C05478=1134.009,150.819,-59.424,-178.763,7.145,148.974
C05479=1134.004,151.068,-59.444,-178.760,7.148,148.974
C05480=1133.999,151.317,-59.466,-178.758,7.150,148.974
C05481=1133.994,151.566,-59.487,-178.755,7.152,148.973
C05482=1133.989,151.815,-59.509,-178.752,7.154,148.973
C05483=1133.985,152.064,-59.529,-178.749,7.156,148.973
C05484=1133.980,152.313,-59.551,-178.746,7.158,148.972
C05485=1133.975,152.562,-59.572,-178.744,7.160,148.972
C05486=1133.970,152.811,-59.594,-178.741,7.162,148.972
C05487=1133.966,153.061,-59.615,-178.738,7.165,148.971
C05488=1133.962,153.309,-59.636,-178.735,7.166,148.971
C05489=1133.957,153.558,-59.657,-178.732,7.168,148.971
C05490=1133.952,153.807,-59.679,-178.729,7.171,148.970
C05491=1133.947,154.057,-59.700,-178.727,7.173,148.970
C05492=1133.942,154.306,-59.722,-178.723,7.175,148.970
C05493=1133.938,154.554,-59.743,-178.721,7.177,148.969
C05494=1133.934,154.804,-59.764,-178.718,7.179,148.969
C05495=1133.929,155.053,-59.786,-178.715,7.181,148.969
C05496=1133.923,155.302,-59.807,-178.712,7.183,148.968
C05497=1133.919,155.550,-59.828,-178.709,7.186,148.968
C05498=1133.914,155.800,-59.851,-178.707,7.188,148.968
C05499=1133.909,156.049,-59.871,-178.704,7.189,148.967
C05500=1133.904,156.298,-59.893,-178.701,7.192,148.967
C05501=1133.900,156.547,-59.915,-178.698,7.194,148.967
C05502=1133.896,156.795,-59.936,-178.695,7.196,148.967
C05503=1133.890,157.065,-59.960,-178.692,7.198,148.966
C05504=1133.885,157.334,-59.983,-178.689,7.201,148.966
C05505=1133.881,157.603,-60.006,-178.686,7.203,148.965
C05506=1133.875,157.872,-60.030,-178.683,7.205,148.965
C05507=1133.870,158.121,-60.052,-178.680,7.207,148.965
C05508=1133.866,158.371,-60.073,-178.678,7.209,148.965
C05509=1133.861,158.619,-60.095,-178.675,7.211,148.964
C05510=1133.856,158.868,-60.116,-178.672,7.214,148.964
C05511=1133.852,159.117,-60.138,-178.669,7.215,148.963
C05512=1133.847,159.366,-60.160,-178.666,7.218,148.963
C05513=1133.842,159.615,-60.182,-178.663,7.220,148.963
C05514=1133.838,159.864,-60.204,-178.660,7.223,148.963
C05515=1133.832,160.113,-60.225,-178.658,7.225,148.962
C05516=1133.828,160.362,-60.247,-178.655,7.226,148.962
C05517=1133.823,160.611,-60.268,-178.652,7.229,148.962
C05518=1133.819,160.860,-60.290,-178.649,7.231,148.961
C05519=1133.814,161.109,-60.312,-178.646,7.233,148.961
C05520=1133.810,161.358,-60.334,-178.643,7.235,148.961
C05521=1133.805,161.607,-60.356,-178.640,7.238,148.960
C05522=1133.800,161.856,-60.378,-178.638,7.240,148.960
C05523=1133.796,162.105,-60.400,-178.635,7.241,148.960
C05524=1133.791,162.354,-60.421,-178.632,7.244,148.959
C05525=1133.787,162.603,-60.443,-178.629,7.246,148.959
C05526=1133.782,162.852,-60.465,-178.626,7.248,148.959
C05527=1133.778,163.101,-60.487,-178.624,7.250,148.959
C05528=1133.772,163.350,-60.509,-178.620,7.253,148.958
C05529=1133.768,163.599,-60.531,-178.618,7.255,148.958
C05530=1133.763,163.848,-60.553,-178.615,7.257,148.958
C05531=1133.759,164.097,-60.575,-178.612,7.259,148.957
C05532=1133.754,164.346,-60.597,-178.609,7.262,148.957
C05533=1133.749,164.595,-60.619,-178.607,7.264,148.957
C05534=1133.745,164.844,-60.641,-178.604,7.265,148.956
C05535=1133.740,165.093,-60.664,-178.601,7.268,148.956
C05536=1133.735,165.341,-60.686,-178.598,7.270,148.956
C05537=1133.731,165.591,-60.708,-178.595,7.272,148.956
C05538=1133.726,165.839,-60.729,-178.593,7.274,148.955
C05539=1133.721,166.089,-60.752,-178.589,7.277,148.955
C05540=1133.716,166.338,-60.774,-178.587,7.279,148.955
C05541=1133.712,166.586,-60.796,-178.584,7.282,148.955
C05542=1133.707,166.835,-60.818,-178.581,7.283,148.954
C05543=1133.702,167.085,-60.841,-178.578,7.286,148.954
C05544=1133.698,167.334,-60.863,-178.576,7.288,148.954
C05545=1133.693,167.583,-60.884,-178.572,7.290,148.953
C05546=1133.689,167.831,-60.907,-178.570,7.292,148.953
C05547=1133.683,168.080,-60.929,-178.567,7.295,148.953
C05548=1133.679,168.330,-60.952,-178.564,7.297,148.952
C05549=1133.675,168.578,-60.974,-178.561,7.299,148.952
C05550=1133.670,168.827,-60.997,-178.559,7.301,148.952
C05551=1133.665,169.077,-61.019,-178.555,7.304,148.952
C05552=1133.661,169.325,-61.041,-178.553,7.306,148.951
C05553=1133.656,169.574,-61.064,-178.550,7.308,148.951
C05554=1133.651,169.823,-61.085,-178.547,7.310,148.951
C05555=1133.647,170.072,-61.108,-178.544,7.313,148.950
C05556=1133.642,170.321,-61.131,-178.542,7.315,148.950
C05557=1133.637,170.570,-61.152,-178.538,7.317,148.950
C05558=1133.633,170.819,-61.175,-178.536,7.319,148.950
C05559=1133.627,171.068,-61.197,-178.533,7.322,148.949
C05560=1133.624,171.316,-61.220,-178.530,7.324,148.949
C05561=1133.619,171.566,-61.243,-178.527,7.326,148.949
C05562=1133.614,171.814,-61.265,-178.524,7.328,148.948
C05563=1133.610,172.064,-61.287,-178.521,7.331,148.948
C05564=1133.605,172.313,-61.310,-178.519,7.333,148.948
C05565=1133.600,172.561,-61.332,-178.516,7.335,148.948
C05566=1133.595,172.811,-61.355,-178.513,7.337,148.947
C05567=1133.591,173.060,-61.378,-178.510,7.340,148.947
C05568=1133.586,173.308,-61.401,-178.507,7.342,148.947
C05569=1133.582,173.557,-61.423,-178.505,7.344,148.947
C05570=1133.577,173.806,-61.446,-178.501,7.347,148.946
C05571=1133.572,174.055,-61.468,-178.499,7.349,148.946
C05572=1133.567,174.304,-61.491,-178.496,7.352,148.946
C05573=1133.563,174.553,-61.513,-178.493,7.353,148.945
C05574=1133.558,174.802,-61.537,-178.490,7.356,148.945
C05575=1133.554,175.050,-61.559,-178.487,7.358,148.945
C05576=1133.549,175.300,-61.582,-178.485,7.361,148.945
C05577=1133.545,175.549,-61.604,-178.482,7.362,148.944
C05578=1133.540,175.798,-61.628,-178.479,7.365,148.944
C05579=1133.535,176.046,-61.649,-178.476,7.368,148.944
C05580=1133.531,176.295,-61.673,-178.473,7.370,148.944
C05581=1133.527,176.544,-61.696,-178.470,7.372,148.943
C05582=1133.522,176.794,-61.718,-178.468,7.374,148.943
C05583=1133.516,177.042,-61.741,-178.464,7.377,148.943
C05584=1133.512,177.291,-61.764,-178.462,7.379,148.943
C05585=1133.507,177.540,-61.787,-178.459,7.381,148.942
C05586=1133.503,177.789,-61.809,-178.456,7.384,148.942
C05587=1133.498,178.038,-61.832,-178.453,7.386,148.942
C05588=1133.493,178.287,-61.856,-178.450,7.389,148.942
C05589=1133.489,178.535,-61.879,-178.448,7.391,148.941
C05590=1133.484,178.785,-61.901,-178.445,7.393,148.941
C05591=1133.481,179.020,-61.923,-178.442,7.395,148.941
C05592=1133.476,179.256,-61.945,-178.439,7.398,148.941
C05593=1133.471,179.491,-61.967,-178.437,7.400,148.940
C05594=1133.449,180.668,-62.075,-179.293,9.081,149.576
C05595=1133.445,180.917,-62.098,-179.289,9.084,149.576
C05596=1133.440,181.165,-62.123,-179.286,9.087,149.576
C05597=1133.435,181.415,-62.146,-179.283,9.091,149.575
C05598=1133.431,181.664,-62.169,-179.280,9.094,149.575
C05599=1133.427,181.912,-62.192,-179.277,9.098,149.576
C05600=1133.422,182.161,-62.216,-179.274,9.100,149.575
C05601=1133.418,182.410,-62.239,-179.271,9.104,149.575
C05602=1133.413,182.659,-62.263,-179.268,9.107,149.575
C05603=1133.409,182.907,-62.287,-179.266,9.110,149.575
C05604=1133.404,183.156,-62.310,-179.262,9.114,149.575
C05605=1133.399,183.405,-62.334,-179.259,9.117,149.575
C05606=1133.395,183.654,-62.358,-179.257,9.120,149.575
C05607=1133.391,183.903,-62.381,-179.254,9.123,149.575
C05608=1133.386,184.152,-62.405,-179.251,9.127,149.575
C05609=1133.382,184.401,-62.429,-179.248,9.130,149.575
C05610=1133.377,184.650,-62.452,-179.246,9.133,149.575
C05611=1133.370,184.985,-62.485,-179.243,9.137,149.575
C05612=1133.364,185.319,-62.516,-179.238,9.141,149.575
C05613=1133.358,185.653,-62.548,-179.235,9.145,149.575
C05614=1133.352,185.987,-62.581,-179.232,9.149,149.575
C05615=1133.347,186.236,-62.604,-179.230,9.152,149.575
C05616=1133.343,186.485,-62.628,-179.227,9.154,149.575
C05617=1133.339,186.734,-62.652,-179.224,9.158,149.575
C05618=1133.334,186.983,-62.676,-179.222,9.161,149.575
C05619=1133.329,187.232,-62.700,-179.220,9.163,149.575
C05620=1133.325,187.481,-62.724,-179.217,9.166,149.575
C05621=1133.320,187.730,-62.747,-179.215,9.169,149.575
C05622=1133.315,187.978,-62.771,-179.212,9.172,149.575
C05623=1133.311,188.226,-62.795,-179.210,9.175,149.575
C05624=1133.306,188.475,-62.819,-179.208,9.178,149.575
C05625=1133.302,188.725,-62.844,-179.206,9.180,149.575
C05626=1133.297,188.974,-62.867,-179.203,9.183,149.575
C05627=1133.293,189.222,-62.891,-179.201,9.186,149.576
C05628=1133.288,189.471,-62.915,-179.199,9.189,149.576
C05629=1133.284,189.720,-62.939,-179.197,9.191,149.576
C05630=1133.279,189.968,-62.963,-179.194,9.194,149.576
C05631=1133.275,190.218,-62.988,-179.192,9.196,149.576
C05632=1133.270,190.466,-63.012,-179.191,9.199,149.576
C05633=1133.266,190.715,-63.035,-179.188,9.202,149.576
C05634=1133.261,190.964,-63.060,-179.187,9.205,149.576
C05635=1133.256,191.212,-63.084,-179.185,9.207,149.576
C05636=1133.251,191.461,-63.107,-179.183,9.210,149.576
C05637=1133.248,191.710,-63.132,-179.181,9.213,149.576
C05638=1133.243,191.959,-63.156,-179.179,9.215,149.576
C05639=1133.238,192.207,-63.180,-179.177,9.218,149.577
C05640=1133.234,192.456,-63.204,-179.175,9.220,149.577
C05641=1133.229,192.706,-63.229,-179.174,9.222,149.577
C05642=1133.224,192.954,-63.253,-179.172,9.225,149.577
C05643=1133.220,193.203,-63.277,-179.170,9.227,149.577
C05644=1133.215,193.451,-63.302,-179.169,9.230,149.577
C05645=1133.211,193.700,-63.326,-179.167,9.232,149.577
C05646=1133.206,193.950,-63.349,-179.165,9.235,149.577
C05647=1133.201,194.198,-63.374,-179.164,9.238,149.578
C05648=1133.197,194.447,-63.398,-179.162,9.240,149.578
C05649=1133.193,194.695,-63.422,-179.161,9.243,149.578
C05650=1133.188,194.945,-63.447,-179.159,9.246,149.578
C05651=1133.184,195.193,-63.471,-179.158,9.247,149.578
C05652=1133.179,195.441,-63.495,-179.156,9.250,149.578
C05653=1133.174,195.690,-63.520,-179.155,9.253,149.579
C05654=1133.170,195.939,-63.544,-179.153,9.255,149.579
C05655=1133.166,196.188,-63.568,-179.153,9.257,149.579
C05656=1133.160,196.437,-63.593,-179.148,9.261,149.579
C05657=1133.157,196.686,-63.617,-179.144,9.266,149.579
C05658=1133.152,196.935,-63.642,-179.140,9.269,149.579
C05659=1133.147,197.183,-63.666,-179.136,9.273,149.578
C05660=1133.143,197.432,-63.690,-179.132,9.277,149.578
C05661=1133.138,197.681,-63.715,-179.128,9.281,149.578
C05662=1133.134,197.929,-63.739,-179.123,9.285,149.578
C05663=1133.129,198.144,-63.761,-179.120,9.288,149.578
C05664=1133.126,198.358,-63.782,-179.117,9.291,149.577
C05665=1133.122,198.572,-63.803,-179.113,9.295,149.577
C05666=1133.118,198.787,-63.824,-179.110,9.298,149.577
C05667=1133.115,199.002,-63.845,-179.107,9.301,149.577
C05668=1133.110,199.216,-63.867,-179.103,9.304,149.577
C05669=1133.106,199.431,-63.888,-179.100,9.307,149.577
C05670=1133.103,199.645,-63.909,-179.097,9.311,149.577
C05671=1133.098,199.894,-63.934,-179.093,9.314,149.576
C05672=1133.094,200.143,-63.959,-179.089,9.318,149.576
C05673=1133.089,200.392,-63.983,-179.085,9.321,149.576
C05674=1133.085,200.639,-64.008,-179.082,9.324,149.576
C05675=1133.080,200.889,-64.033,-179.078,9.328,149.576
C05676=1133.075,201.138,-64.058,-179.075,9.331,149.576
C05677=1133.071,201.387,-64.082,-179.071,9.335,149.575
C05678=1133.066,201.635,-64.108,-179.068,9.338,149.575
C05679=1133.063,201.884,-64.132,-179.065,9.341,149.575
C05680=1133.058,202.133,-64.157,-179.061,9.345,149.575
C05681=1133.053,202.381,-64.182,-179.058,9.347,149.575
C05682=1133.049,202.630,-64.206,-179.054,9.351,149.575
C05683=1133.045,202.879,-64.232,-179.051,9.354,149.575
C05684=1133.040,203.127,-64.257,-179.048,9.357,149.574
C05685=1133.035,203.376,-64.281,-179.045,9.360,149.574
C05686=1133.031,203.625,-64.307,-179.041,9.363,149.574
C05687=1133.026,203.873,-64.331,-179.038,9.366,149.574
C05688=1133.022,204.122,-64.357,-179.035,9.369,149.574
C05689=1133.017,204.370,-64.381,-179.033,9.372,149.574
C05690=1133.013,204.619,-64.407,-179.029,9.375,149.574
C05691=1133.008,204.868,-64.432,-179.026,9.378,149.574
C05692=1133.004,205.117,-64.457,-179.023,9.381,149.573
C05693=1133.000,205.366,-64.482,-179.020,9.384,149.573
C05694=1132.995,205.614,-64.507,-179.018,9.387,149.573
C05695=1132.990,205.863,-64.532,-179.015,9.390,149.573
C05696=1132.986,206.112,-64.558,-179.012,9.392,149.573
C05697=1132.981,206.360,-64.583,-179.010,9.395,149.573
C05698=1132.976,206.609,-64.608,-179.007,9.397,149.573
C05699=1132.973,206.858,-64.633,-179.005,9.401,149.573
C05700=1132.968,207.106,-64.658,-179.002,9.403,149.573
C05701=1132.963,207.355,-64.684,-179.000,9.406,149.573
C05702=1132.959,207.604,-64.709,-178.997,9.408,149.573
C05703=1132.954,207.853,-64.734,-178.995,9.411,149.573
C05704=1132.950,208.101,-64.760,-178.992,9.414,149.573
C05705=1132.945,208.350,-64.785,-178.991,9.416,149.573
C05706=1132.940,208.599,-64.810,-178.988,9.419,149.573
C05707=1132.936,208.847,-64.835,-178.986,9.421,149.573
C05708=1132.932,209.096,-64.861,-178.984,9.423,149.573
C05709=1132.928,209.344,-64.886,-178.981,9.427,149.573
C05710=1132.923,209.593,-64.911,-178.979,9.429,149.573
C05711=1132.919,209.842,-64.937,-178.978,9.431,149.573
C05712=1132.914,210.091,-64.963,-178.976,9.434,149.573
C05713=1132.910,210.339,-64.988,-178.974,9.436,149.573
C05714=1132.905,210.588,-65.013,-178.972,9.439,149.573
C05715=1132.900,210.836,-65.038,-178.970,9.441,149.573
C05716=1132.896,211.085,-65.064,-178.968,9.443,149.573
C05717=1132.892,211.334,-65.090,-178.967,9.446,149.574
C05718=1132.887,211.582,-65.115,-178.965,9.448,149.574
C05719=1132.884,211.797,-65.137,-178.963,9.451,149.574
C05720=1132.880,212.011,-65.159,-178.962,9.453,149.574
C05721=1132.875,212.225,-65.181,-178.960,9.455,149.574
C05722=1132.872,212.440,-65.203,-178.960,9.457,149.574
C05723=1132.868,212.654,-65.225,-178.958,9.458,149.574
C05724=1132.864,212.868,-65.247,-178.957,9.461,149.575
C05725=1132.860,213.083,-65.269,-178.956,9.463,149.575
C05726=1132.856,213.297,-65.291,-178.955,9.465,149.575
C05727=1132.852,213.546,-65.317,-178.953,9.467,149.575
C05728=1132.847,213.794,-65.342,-178.952,9.470,149.575
C05729=1132.843,214.043,-65.368,-178.950,9.472,149.575
C05730=1132.839,214.292,-65.394,-178.948,9.476,149.576
C05731=1132.834,214.540,-65.419,-178.946,9.478,149.576
C05732=1132.830,214.789,-65.445,-178.944,9.481,149.576
C05733=1132.825,215.038,-65.471,-178.943,9.483,149.576
C05734=1132.821,215.286,-65.496,-178.940,9.487,149.576
C05735=1132.816,215.535,-65.522,-178.939,9.489,149.576
C05736=1132.812,215.783,-65.548,-178.937,9.492,149.576
C05737=1132.808,216.032,-65.573,-178.935,9.495,149.577
C05738=1132.803,216.280,-65.599,-178.933,9.497,149.577
C05739=1132.799,216.529,-65.625,-178.931,9.501,149.577
C05740=1132.795,216.778,-65.650,-178.929,9.503,149.577
C05741=1132.790,217.026,-65.676,-178.927,9.506,149.577
C05742=1132.785,217.275,-65.702,-178.925,9.509,149.577
C05743=1132.781,217.524,-65.728,-178.922,9.512,149.577
C05744=1132.776,217.773,-65.754,-178.920,9.515,149.577
C05745=1132.772,218.021,-65.779,-178.918,9.518,149.578
C05746=1132.767,218.270,-65.805,-178.916,9.521,149.578
C05747=1132.763,218.518,-65.830,-178.914,9.524,149.578
C05748=1132.759,218.767,-65.856,-178.911,9.527,149.578
C05749=1132.754,219.016,-65.883,-178.908,9.530,149.578
C05750=1132.749,219.264,-65.909,-178.906,9.533,149.578
C05751=1132.745,219.513,-65.934,-178.903,9.537,149.578
C05752=1132.741,219.761,-65.960,-178.901,9.540,149.578
C05753=1132.737,220.010,-65.986,-178.898,9.543,149.578
C05754=1132.732,220.259,-66.012,-178.896,9.546,149.578
C05755=1132.727,220.507,-66.038,-178.893,9.549,149.578
C05756=1132.723,220.756,-66.064,-178.891,9.552,149.578
C05757=1132.719,221.004,-66.090,-178.888,9.555,149.578
C05758=1132.714,221.254,-66.116,-178.886,9.558,149.579
C05759=1132.710,221.502,-66.142,-178.883,9.561,149.579
C05760=1132.705,221.750,-66.168,-178.880,9.565,149.579
C05761=1132.701,221.999,-66.194,-178.877,9.568,149.579
C05762=1132.696,222.248,-66.220,-178.875,9.572,149.579
C05763=1132.692,222.496,-66.247,-178.872,9.575,149.579
C05764=1132.688,222.745,-66.272,-178.869,9.578,149.579
C05765=1132.683,222.994,-66.299,-178.866,9.581,149.579
C05766=1132.679,223.242,-66.325,-178.863,9.585,149.579
C05767=1132.674,223.490,-66.351,-178.860,9.588,149.579
C05768=1132.669,223.739,-66.378,-178.857,9.592,149.579
C05769=1132.665,223.987,-66.403,-178.855,9.595,149.579
C05770=1132.661,224.236,-66.429,-178.851,9.598,149.579
C05771=1132.656,224.485,-66.456,-178.848,9.601,149.579
C05772=1132.652,224.734,-66.482,-178.845,9.605,149.579
C05773=1132.648,224.982,-66.508,-178.842,9.609,149.579
C05774=1132.643,225.231,-66.535,-178.838,9.612,149.579
C05775=1132.639,225.445,-66.558,-178.836,9.616,149.579
C05776=1132.636,225.659,-66.581,-178.833,9.618,149.579
C05777=1132.631,225.873,-66.603,-178.830,9.621,149.578
C05778=1132.628,226.088,-66.626,-178.827,9.624,149.578
C05779=1132.624,226.301,-66.649,-178.824,9.627,149.578
C05780=1132.620,226.516,-66.671,-178.821,9.630,149.578
C05781=1132.616,226.730,-66.694,-178.818,9.633,149.578
C05782=1132.613,226.944,-66.717,-178.815,9.636,149.578
C05783=1132.608,227.193,-66.743,-178.812,9.640,149.578
C05784=1132.604,227.441,-66.770,-178.808,9.643,149.578
C05785=1132.600,227.690,-66.796,-178.804,9.647,149.578
C05786=1132.595,227.939,-66.823,-178.801,9.650,149.578
C05787=1132.591,228.187,-66.849,-178.797,9.654,149.578
C05788=1132.586,228.435,-66.876,-178.794,9.657,149.577
C05789=1132.582,228.684,-66.902,-178.790,9.661,149.577
C05790=1132.577,228.933,-66.929,-178.786,9.664,149.577
C05791=1132.573,229.181,-66.956,-178.782,9.668,149.577
C05792=1132.569,229.429,-66.983,-178.778,9.672,149.577
C05793=1132.564,229.679,-67.009,-178.775,9.675,149.577
C05794=1132.560,229.927,-67.035,-178.771,9.679,149.576
C05795=1132.555,230.175,-67.062,-178.766,9.683,149.576
C05796=1132.551,230.424,-67.089,-178.762,9.686,149.576
C05797=1132.547,230.672,-67.116,-178.759,9.690,149.576
C05798=1132.542,230.920,-67.143,-178.755,9.693,149.576
C05799=1132.537,231.169,-67.170,-178.751,9.696,149.575
C05800=1132.534,231.418,-67.197,-178.748,9.700,149.575
C05801=1132.529,231.667,-67.223,-178.745,9.702,149.575
C05802=1132.524,231.915,-67.250,-178.741,9.706,149.575
C05803=1132.521,232.164,-67.277,-178.737,9.709,149.575
C05804=1132.516,232.412,-67.304,-178.734,9.713,149.575
C05805=1132.511,232.661,-67.331,-178.731,9.715,149.575
C05806=1132.507,232.909,-67.358,-178.727,9.719,149.574
C05807=1132.503,233.157,-67.384,-178.724,9.721,149.574
C05808=1132.499,233.406,-67.412,-178.720,9.725,149.574
C05809=1132.494,233.654,-67.440,-178.717,9.728,149.574
C05810=1132.490,233.903,-67.467,-178.714,9.731,149.574
C05811=1132.486,234.151,-67.493,-178.711,9.734,149.574
C05812=1132.481,234.399,-67.520,-178.708,9.737,149.573
C05813=1132.476,234.648,-67.547,-178.704,9.740,149.573
C05814=1132.472,234.897,-67.575,-178.701,9.742,149.573
C05815=1132.468,235.146,-67.602,-178.698,9.745,149.573
C05816=1132.463,235.394,-67.629,-178.695,9.748,149.573
C05817=1132.459,235.642,-67.656,-178.692,9.751,149.573
C05818=1132.455,235.890,-67.683,-178.689,9.753,149.573
C05819=1132.451,236.139,-67.711,-178.686,9.756,149.572
C05820=1132.446,236.388,-67.738,-178.683,9.759,149.572
C05821=1132.441,236.636,-67.765,-178.681,9.762,149.572
C05822=1132.437,236.884,-67.792,-178.678,9.765,149.572
C05823=1132.433,237.133,-67.820,-178.675,9.768,149.572
C05824=1132.428,237.382,-67.847,-178.672,9.770,149.572
C05825=1132.424,237.630,-67.875,-178.669,9.772,149.572
C05826=1132.419,237.878,-67.902,-178.666,9.775,149.572
C05827=1132.416,238.127,-67.929,-178.665,9.777,149.572
C05828=1132.411,238.376,-67.956,-178.662,9.780,149.572
C05829=1132.407,238.624,-67.983,-178.659,9.782,149.571
C05830=1132.402,238.872,-68.010,-178.657,9.785,149.572
C05831=1132.398,239.086,-68.035,-178.654,9.787,149.571
C05832=1132.395,239.301,-68.058,-178.653,9.790,149.571
C05833=1132.391,239.515,-68.082,-178.650,9.791,149.571
C05834=1132.387,239.728,-68.105,-178.648,9.794,149.571
C05835=1132.383,239.943,-68.129,-178.647,9.795,149.571
C05836=1132.380,240.157,-68.153,-178.645,9.797,149.571
C05837=1132.376,240.371,-68.176,-178.643,9.800,149.571
C05838=1132.372,240.585,-68.201,-178.641,9.802,149.571
C05839=1132.368,240.834,-68.228,-178.639,9.804,149.571
C05840=1132.363,241.082,-68.255,-178.637,9.806,149.571
C05841=1132.359,241.331,-68.283,-178.634,9.808,149.571
C05842=1132.355,241.579,-68.310,-178.633,9.811,149.571
C05843=1132.350,241.827,-68.338,-178.631,9.813,149.571
C05844=1132.346,242.076,-68.365,-178.629,9.815,149.571
C05845=1132.342,242.324,-68.393,-178.627,9.818,149.571
C05846=1132.337,242.573,-68.420,-178.625,9.820,149.571
C05847=1132.334,242.821,-68.448,-178.623,9.822,149.572
C05848=1132.329,243.070,-68.475,-178.622,9.824,149.572
C05849=1132.325,243.317,-68.503,-178.620,9.826,149.572
C05850=1132.320,243.567,-68.531,-178.618,9.828,149.572
C05851=1132.315,243.815,-68.559,-178.617,9.830,149.572
C05852=1132.311,244.063,-68.587,-178.615,9.832,149.572
C05853=1132.307,244.312,-68.614,-178.613,9.835,149.572
C05854=1132.303,244.560,-68.642,-178.612,9.837,149.572
C05855=1132.298,244.808,-68.669,-178.610,9.839,149.572
C05856=1132.294,245.057,-68.697,-178.609,9.841,149.572
C05857=1132.290,245.305,-68.725,-178.607,9.843,149.572
C05858=1132.286,245.554,-68.752,-178.606,9.845,149.572
C05859=1132.281,245.802,-68.781,-178.605,9.847,149.573
C05860=1132.276,246.051,-68.808,-178.604,9.849,149.573
C05861=1132.272,246.299,-68.836,-178.603,9.851,149.573
C05862=1132.268,246.547,-68.863,-178.602,9.853,149.573
C05863=1132.263,246.796,-68.891,-178.601,9.855,149.573
C05864=1132.260,247.044,-68.919,-178.599,9.857,149.574
C05865=1132.254,247.292,-68.947,-178.598,9.859,149.574
C05866=1132.250,247.542,-68.974,-178.594,9.863,149.574
C05867=1132.246,247.789,-69.002,-178.586,9.869,149.573
C05868=1132.242,248.037,-69.030,-178.578,9.875,149.572
C05869=1132.238,248.286,-69.057,-178.571,9.880,149.572
C05870=1132.233,248.535,-69.086,-178.565,9.886,149.571
C05871=1132.229,248.783,-69.114,-178.557,9.891,149.571
C05872=1132.224,249.031,-69.142,-178.551,9.895,149.570
C05873=1132.221,249.280,-69.170,-178.545,9.900,149.569
C05874=1132.216,249.528,-69.198,-178.539,9.905,149.569
C05875=1132.212,249.776,-69.226,-178.533,9.909,149.569
C05876=1132.207,250.025,-69.255,-178.528,9.913,149.568
C05877=1132.203,250.273,-69.283,-178.523,9.917,149.568
C05878=1132.199,250.521,-69.311,-178.518,9.920,149.567
C05879=1132.194,250.770,-69.339,-178.513,9.924,149.567
C05880=1132.190,251.018,-69.367,-178.509,9.928,149.567
C05881=1132.185,251.267,-69.396,-178.505,9.931,149.566
C05882=1132.182,251.515,-69.424,-178.501,9.934,149.566
C05883=1132.177,251.763,-69.452,-178.498,9.936,149.566
C05884=1132.173,252.012,-69.481,-178.495,9.939,149.566
C05885=1132.168,252.260,-69.508,-178.491,9.942,149.565
C05886=1132.164,252.509,-69.537,-178.489,9.943,149.565
C05887=1132.160,252.723,-69.562,-178.487,9.945,149.565
C05888=1132.157,252.936,-69.586,-178.485,9.948,149.565
C05889=1132.153,253.150,-69.611,-178.483,9.949,149.565
C05890=1132.149,253.364,-69.635,-178.482,9.951,149.565
C05891=1132.146,253.578,-69.660,-178.481,9.952,149.565
C05892=1132.142,253.792,-69.684,-178.480,9.953,149.565
C05893=1132.138,254.006,-69.709,-178.479,9.954,149.565
C05894=1132.134,254.220,-69.733,-178.479,9.956,149.565
C05895=1132.131,254.468,-69.762,-178.478,9.956,149.565
C05896=1132.125,254.716,-69.790,-178.478,9.957,149.566
C05897=1132.122,254.965,-69.818,-178.479,9.958,149.566
C05898=1132.117,255.214,-69.847,-178.478,9.959,149.566
C05899=1132.113,255.462,-69.875,-178.479,9.960,149.567
C05900=1132.109,255.710,-69.904,-178.481,9.960,149.567
C05901=1132.104,255.958,-69.932,-178.481,9.961,149.567
C05902=1132.100,256.207,-69.961,-178.479,9.963,149.567
C05903=1132.096,256.455,-69.989,-178.476,9.966,149.567
C05904=1132.091,256.704,-70.017,-178.473,9.969,149.567
C05905=1132.088,256.952,-70.046,-178.470,9.972,149.567
C05906=1132.083,257.200,-70.075,-178.467,9.976,149.567
C05907=1132.078,257.449,-70.103,-178.464,9.978,149.567
C05908=1132.074,257.697,-70.131,-178.461,9.981,149.567
C05909=1132.069,257.945,-70.161,-178.458,9.984,149.567
C05910=1132.066,258.193,-70.189,-178.454,9.987,149.567
C05911=1132.061,258.442,-70.217,-178.451,9.990,149.566
C05912=1132.057,258.689,-70.246,-178.448,9.993,149.566
C05913=1132.053,258.938,-70.275,-178.444,9.996,149.566
C05914=1132.049,259.187,-70.304,-178.441,9.999,149.566
C05915=1132.045,259.435,-70.332,-178.438,10.002,149.566
C05916=1132.040,259.683,-70.361,-178.435,10.005,149.566
C05917=1132.036,259.932,-70.390,-178.431,10.008,149.565
C05918=1132.032,260.180,-70.418,-178.428,10.011,149.565
C05919=1132.027,260.428,-70.447,-178.424,10.015,149.565
C05920=1132.022,260.677,-70.476,-178.421,10.017,149.565
C05921=1132.019,260.925,-70.505,-178.417,10.021,149.565
C05922=1132.015,261.174,-70.534,-178.414,10.024,149.565
C05923=1132.010,261.421,-70.563,-178.410,10.026,149.564
C05924=1132.005,261.670,-70.591,-178.407,10.030,149.564
C05925=1132.002,261.918,-70.620,-178.403,10.033,149.564
C05926=1131.997,262.167,-70.649,-178.399,10.036,149.564
C05927=1131.993,262.414,-70.678,-178.396,10.039,149.564
C05928=1131.988,262.663,-70.708,-178.392,10.042,149.563
C05929=1131.985,262.911,-70.736,-178.388,10.045,149.563
C05930=1131.980,263.160,-70.765,-178.384,10.049,149.563
C05931=1131.975,263.408,-70.794,-178.380,10.052,149.563
C05932=1131.971,263.656,-70.823,-178.376,10.055,149.562
C05933=1131.967,263.904,-70.852,-178.372,10.058,149.562
C05934=1131.963,264.152,-70.882,-178.368,10.062,149.562
C05935=1131.959,264.401,-70.910,-178.364,10.065,149.562
C05936=1131.954,264.649,-70.939,-178.361,10.068,149.562
C05937=1131.950,264.897,-70.969,-178.359,10.070,149.561
C05938=1131.946,265.145,-70.998,-178.357,10.072,149.561
C05939=1131.941,265.394,-71.027,-178.354,10.074,149.561
C05940=1131.937,265.642,-71.056,-178.352,10.077,149.561
C05941=1131.933,265.891,-71.086,-178.350,10.079,149.561
C05942=1131.928,266.138,-71.115,-178.347,10.081,149.561
C05943=1131.925,266.353,-71.140,-178.344,10.083,149.561
C05944=1131.921,266.566,-71.165,-178.343,10.086,149.561
C05945=1131.918,266.780,-71.190,-178.341,10.087,149.561
C05946=1131.914,266.993,-71.216,-178.339,10.089,149.561
C05947=1131.910,267.208,-71.241,-178.336,10.091,149.561
C05948=1131.907,267.422,-71.266,-178.334,10.093,149.561
C05949=1131.903,267.635,-71.291,-178.332,10.095,149.560
C05950=1131.899,267.849,-71.317,-178.329,10.098,149.560
C05951=1131.894,268.098,-71.345,-178.327,10.100,149.560
C05952=1131.890,268.346,-71.375,-178.324,10.103,149.560
C05953=1131.886,268.594,-71.404,-178.322,10.105,149.560
C05954=1131.882,268.843,-71.434,-178.319,10.107,149.560
C05955=1131.878,269.091,-71.463,-178.317,10.110,149.560
C05956=1131.873,269.339,-71.493,-178.314,10.113,149.560
C05957=1131.869,269.587,-71.522,-178.311,10.115,149.560
C05958=1131.865,269.836,-71.552,-178.308,10.118,149.560
C05959=1131.861,270.084,-71.581,-178.306,10.120,149.560
C05960=1131.857,270.332,-71.611,-178.303,10.123,149.559
C05961=1131.853,270.580,-71.640,-178.300,10.126,149.559
C05962=1131.848,270.828,-71.669,-178.297,10.128,149.559
C05963=1131.844,271.076,-71.699,-178.295,10.130,149.559
C05964=1131.839,271.324,-71.728,-178.292,10.133,149.559
C05965=1131.836,271.572,-71.758,-178.289,10.136,149.559
C05966=1131.831,271.820,-71.788,-178.286,10.139,149.559
C05967=1131.827,272.069,-71.817,-178.282,10.141,149.559
C05968=1131.823,272.317,-71.847,-178.279,10.144,149.558
C05969=1131.819,272.565,-71.876,-178.276,10.146,149.558
C05970=1131.814,272.814,-71.906,-178.274,10.148,149.558
C05971=1131.810,273.062,-71.936,-178.271,10.151,149.558
C05972=1131.806,273.310,-71.966,-178.268,10.154,149.558
C05973=1131.802,273.558,-71.995,-178.265,10.157,149.558
C05974=1131.797,273.806,-72.025,-178.262,10.159,149.558
C05975=1131.793,274.055,-72.054,-178.259,10.162,149.558
C05976=1131.789,274.302,-72.085,-178.255,10.165,149.557
C05977=1131.785,274.551,-72.114,-178.253,10.168,149.557
C05978=1131.780,274.799,-72.144,-178.250,10.171,149.557
C05979=1131.776,275.047,-72.173,-178.246,10.173,149.557
C05980=1131.772,275.295,-72.203,-178.243,10.176,149.557
C05981=1131.768,275.544,-72.234,-178.240,10.179,149.557
C05982=1131.764,275.792,-72.263,-178.237,10.181,149.556
C05983=1131.760,276.040,-72.293,-178.234,10.184,149.556
C05984=1131.756,276.288,-72.323,-178.231,10.188,149.556
C05985=1131.751,276.537,-72.353,-178.227,10.190,149.556
C05986=1131.747,276.785,-72.383,-178.224,10.193,149.556
C05987=1131.743,277.033,-72.412,-178.221,10.195,149.556
C05988=1131.739,277.281,-72.443,-178.217,10.199,149.556
C05989=1131.734,277.529,-72.473,-178.214,10.201,149.555
C05990=1131.730,277.777,-72.502,-178.211,10.204,149.555
C05991=1131.726,278.025,-72.532,-178.207,10.207,149.555
C05992=1131.722,278.274,-72.563,-178.204,10.210,149.555
C05993=1131.718,278.522,-72.593,-178.201,10.212,149.554
C05994=1131.714,278.770,-72.622,-178.197,10.216,149.554
C05995=1131.709,279.018,-72.653,-178.194,10.218,149.554
C05996=1131.705,279.266,-72.683,-178.190,10.221,149.554
C05997=1131.701,279.514,-72.713,-178.187,10.224,149.554
C05998=1131.696,279.762,-72.744,-178.184,10.227,149.553
C05999=1131.693,279.976,-72.769,-178.181,10.229,149.553
C06000=1131.689,280.190,-72.795,-178.177,10.232,149.553
C06001=1131.686,280.404,-72.822,-178.174,10.234,149.553
C06002=1131.682,280.617,-72.847,-178.171,10.237,149.553
C06003=1131.679,280.831,-72.874,-178.168,10.240,149.553
C06004=1131.674,281.045,-72.900,-178.165,10.242,149.552
C06005=1131.672,281.258,-72.926,-178.162,10.244,149.552
C06006=1131.667,281.472,-72.952,-178.159,10.246,149.552
C06007=1131.663,281.720,-72.982,-178.156,10.249,149.552
C06008=1131.659,281.969,-73.012,-178.153,10.252,149.552
C06009=1131.655,282.217,-73.042,-178.150,10.254,149.551
C06010=1131.651,282.464,-73.073,-178.147,10.257,149.551
C06011=1131.647,282.712,-73.103,-178.144,10.260,149.551
C06012=1131.642,282.961,-73.133,-178.140,10.262,149.551
C06013=1131.639,283.209,-73.164,-178.137,10.265,149.551
C06014=1131.634,283.457,-73.195,-178.134,10.267,149.550
C06015=1131.629,283.705,-73.225,-178.131,10.270,149.550
C06016=1131.625,283.953,-73.256,-178.129,10.272,149.550
C06017=1131.621,284.202,-73.286,-178.125,10.274,149.550
C06018=1131.617,284.450,-73.316,-178.122,10.277,149.550
C06019=1131.613,284.697,-73.347,-178.119,10.279,149.550
C06020=1131.609,284.945,-73.377,-178.116,10.282,149.549
C06021=1131.605,285.194,-73.408,-178.113,10.285,149.549
C06022=1131.600,285.442,-73.439,-178.110,10.287,149.549
C06023=1131.596,285.689,-73.469,-178.107,10.290,149.549
C06024=1131.592,285.938,-73.500,-178.104,10.293,149.549
C06025=1131.588,286.186,-73.531,-178.101,10.295,149.549
C06026=1131.584,286.434,-73.561,-178.098,10.297,149.548
C06027=1131.579,286.682,-73.592,-178.095,10.300,149.548
C06028=1131.576,286.930,-73.622,-178.092,10.302,149.548
C06029=1131.571,287.178,-73.653,-178.089,10.305,149.548
C06030=1131.567,287.426,-73.684,-178.085,10.307,149.548
C06031=1131.563,287.674,-73.715,-178.082,10.310,149.547
C06032=1131.559,287.922,-73.745,-178.079,10.313,149.547
C06033=1131.554,288.170,-73.776,-178.076,10.315,149.547
C06034=1131.550,288.419,-73.807,-178.073,10.318,149.547
C06035=1131.546,288.666,-73.837,-178.070,10.320,149.547
C06036=1131.542,288.914,-73.868,-178.067,10.323,149.547
C06037=1131.538,289.163,-73.899,-178.064,10.326,149.546
C06038=1131.533,289.411,-73.930,-178.061,10.328,149.546
C06039=1131.530,289.659,-73.961,-178.058,10.330,149.546
C06040=1131.525,289.907,-73.992,-178.055,10.333,149.546
C06041=1131.521,290.155,-74.023,-178.052,10.335,149.546
C06042=1131.517,290.403,-74.054,-178.049,10.338,149.545
C06043=1131.513,290.651,-74.084,-178.045,10.340,149.545
C06044=1131.509,290.900,-74.115,-178.042,10.343,149.545
C06045=1131.505,291.147,-74.147,-178.040,10.346,149.545
C06046=1131.500,291.395,-74.177,-178.036,10.348,149.545
C06047=1131.496,291.644,-74.209,-178.033,10.351,149.545
C06048=1131.492,291.891,-74.239,-178.030,10.354,149.544
C06049=1131.488,292.139,-74.271,-178.027,10.356,149.544
C06050=1131.484,292.387,-74.301,-178.024,10.358,149.544
C06051=1131.480,292.636,-74.332,-178.021,10.361,149.544
C06052=1131.476,292.883,-74.364,-178.018,10.363,149.544
C06053=1131.471,293.131,-74.395,-178.015,10.366,149.544
C06054=1131.467,293.380,-74.426,-178.012,10.368,149.543
C06055=1131.463,293.594,-74.453,-178.009,10.370,149.543
C06056=1131.460,293.806,-74.480,-178.007,10.373,149.543
C06057=1131.456,294.020,-74.507,-178.004,10.375,149.543
C06058=1131.453,294.234,-74.534,-178.001,10.378,149.543
C06059=1131.449,294.447,-74.560,-177.999,10.380,149.543
C06060=1131.446,294.661,-74.587,-177.996,10.382,149.542
C06061=1131.442,294.875,-74.614,-177.993,10.384,149.542
C06062=1131.439,295.088,-74.641,-177.991,10.386,149.542
C06063=1131.435,295.336,-74.672,-177.988,10.389,149.542
C06064=1131.430,295.584,-74.703,-177.984,10.391,149.542
C06065=1131.426,295.832,-74.735,-177.981,10.394,149.542
C06066=1131.422,296.080,-74.766,-177.978,10.396,149.541
C06067=1131.418,296.328,-74.797,-177.975,10.399,149.541
C06068=1131.414,296.576,-74.829,-177.972,10.401,149.541
C06069=1131.410,296.824,-74.860,-177.969,10.404,149.541
C06070=1131.406,297.072,-74.891,-177.966,10.406,149.541
C06071=1131.401,297.320,-74.923,-177.963,10.409,149.541
C06072=1131.398,297.568,-74.954,-177.960,10.411,149.540
C06073=1131.393,297.816,-74.985,-177.957,10.414,149.540
C06074=1131.389,298.064,-75.017,-177.954,10.416,149.540
C06075=1131.385,298.312,-75.048,-177.951,10.419,149.540
C06076=1131.381,298.560,-75.080,-177.947,10.421,149.540
C06077=1131.377,298.808,-75.112,-177.944,10.424,149.539
C06078=1131.373,299.056,-75.142,-177.941,10.427,149.539
C06079=1131.369,299.304,-75.174,-177.938,10.429,149.539
C06080=1131.365,299.551,-75.206,-177.935,10.432,149.539
C06081=1131.361,299.799,-75.237,-177.931,10.434,149.539
C06082=1131.356,300.048,-75.269,-177.929,10.437,149.539
C06083=1131.352,300.295,-75.301,-177.925,10.439,149.538
C06084=1131.348,300.543,-75.333,-177.923,10.441,149.538
C06085=1131.344,300.791,-75.364,-177.920,10.444,149.538
C06086=1131.340,301.039,-75.395,-177.917,10.447,149.538
C06087=1131.336,301.288,-75.427,-177.913,10.449,149.538
C06088=1131.331,301.535,-75.459,-177.910,10.452,149.537
C06089=1131.327,301.783,-75.491,-177.907,10.454,149.537
C06090=1131.324,302.031,-75.523,-177.904,10.457,149.537
C06091=1131.319,302.279,-75.554,-177.901,10.460,149.537
C06092=1131.315,302.527,-75.585,-177.898,10.462,149.537
C06093=1131.310,302.775,-75.617,-177.895,10.465,149.536
C06094=1131.307,303.023,-75.649,-177.892,10.467,149.536
C06095=1131.303,303.271,-75.681,-177.888,10.470,149.536
C06096=1131.299,303.518,-75.713,-177.885,10.473,149.536
C06097=1131.294,303.767,-75.745,-177.882,10.475,149.536
C06098=1131.290,304.015,-75.777,-177.879,10.478,149.536
C06099=1131.286,304.262,-75.808,-177.876,10.480,149.535
C06100=1131.282,304.510,-75.841,-177.873,10.482,149.535
C06101=1131.278,304.758,-75.873,-177.870,10.485,149.535
C06102=1131.274,305.006,-75.904,-177.867,10.487,149.535
C06103=1131.269,305.254,-75.937,-177.864,10.490,149.535
C06104=1131.265,305.502,-75.968,-177.860,10.492,149.534
C06105=1131.262,305.750,-76.000,-177.858,10.495,149.534
C06106=1131.257,305.998,-76.032,-177.854,10.498,149.534
C06107=1131.253,306.246,-76.064,-177.851,10.500,149.534
C06108=1131.249,306.494,-76.096,-177.848,10.503,149.534
C06109=1131.245,306.742,-76.128,-177.845,10.505,149.533
C06110=1131.241,306.990,-76.160,-177.842,10.508,149.533
C06111=1131.237,307.203,-76.188,-177.839,10.510,149.533
C06112=1131.234,307.416,-76.216,-177.836,10.512,149.533
C06113=1131.231,307.629,-76.243,-177.834,10.514,149.533
C06114=1131.227,307.843,-76.271,-177.831,10.516,149.533
C06115=1131.223,308.057,-76.298,-177.828,10.519,149.533
C06116=1131.219,308.270,-76.326,-177.826,10.521,149.532
C06117=1131.216,308.484,-76.354,-177.823,10.522,149.532
C06118=1131.213,308.697,-76.382,-177.820,10.525,149.532
C06119=1131.209,308.945,-76.414,-177.817,10.528,149.532
C06120=1131.204,309.193,-76.446,-177.814,10.530,149.532
C06121=1131.200,309.440,-76.479,-177.811,10.533,149.532
C06122=1131.197,309.688,-76.511,-177.808,10.536,149.531
C06123=1131.192,309.937,-76.543,-177.804,10.538,149.531
C06124=1131.189,310.184,-76.576,-177.801,10.541,149.531
C06125=1131.184,310.432,-76.608,-177.799,10.542,149.531
C06126=1131.180,310.680,-76.639,-177.796,10.545,149.531
C06127=1131.176,310.927,-76.673,-177.792,10.548,149.530
C06128=1131.172,311.176,-76.705,-177.789,10.550,149.530
C06129=1131.168,311.424,-76.737,-177.786,10.553,149.530
C06130=1131.164,311.671,-76.770,-177.783,10.555,149.530
C06131=1131.159,311.919,-76.802,-177.780,10.558,149.530
C06132=1131.155,312.167,-76.835,-177.777,10.561,149.530
C06133=1131.152,312.415,-76.867,-177.773,10.563,149.529
C06134=1131.147,312.663,-76.899,-177.770,10.566,149.529
C06135=1131.144,312.910,-76.932,-177.767,10.568,149.529
C06136=1131.139,313.159,-76.964,-177.764,10.571,149.529
C06137=1131.135,313.406,-76.997,-177.761,10.573,149.529
C06138=1131.131,313.654,-77.029,-177.757,10.576,149.528
C06139=1131.127,313.902,-77.062,-177.755,10.579,149.528
C06140=1131.123,314.150,-77.094,-177.751,10.581,149.528
C06141=1131.119,314.397,-77.127,-177.748,10.584,149.528
C06142=1131.115,314.645,-77.160,-177.746,10.585,149.528
C06143=1131.111,314.893,-77.192,-177.742,10.588,149.527
C06144=1131.107,315.141,-77.225,-177.739,10.591,149.527
C06145=1131.102,315.389,-77.257,-177.736,10.593,149.527
C06146=1131.099,315.637,-77.290,-177.733,10.596,149.527
C06147=1131.095,315.884,-77.323,-177.730,10.598,149.527
C06148=1131.090,316.133,-77.356,-177.726,10.601,149.527
C06149=1131.087,316.380,-77.388,-177.723,10.604,149.526
C06150=1131.083,316.628,-77.421,-177.720,10.606,149.526
C06151=1131.078,316.876,-77.454,-177.717,10.608,149.526
C06152=1131.074,317.124,-77.487,-177.714,10.611,149.526
C06153=1131.071,317.371,-77.519,-177.711,10.614,149.526
C06154=1131.067,317.619,-77.553,-177.707,10.616,149.525
C06155=1131.062,317.867,-77.585,-177.704,10.619,149.525
C06156=1131.058,318.115,-77.618,-177.701,10.621,149.525
C06157=1131.055,318.362,-77.651,-177.698,10.624,149.525
C06158=1131.051,318.610,-77.684,-177.695,10.627,149.525
C06159=1131.046,318.859,-77.716,-177.691,10.629,149.524
C06160=1131.042,319.106,-77.749,-177.688,10.632,149.524
C06161=1131.038,319.354,-77.783,-177.686,10.633,149.524
C06162=1131.035,319.601,-77.815,-177.682,10.636,149.524
C06163=1131.030,319.849,-77.848,-177.680,10.639,149.524
C06164=1131.026,320.097,-77.881,-177.676,10.641,149.524
C06165=1131.022,320.345,-77.915,-177.673,10.643,149.523
C06166=1131.018,320.592,-77.948,-177.670,10.646,149.523
C06167=1131.014,320.806,-77.976,-177.667,10.649,149.523
C06168=1131.011,321.019,-78.004,-177.664,10.651,149.523
C06169=1131.008,321.233,-78.033,-177.662,10.653,149.523
C06170=1131.004,321.446,-78.061,-177.659,10.655,149.523
C06171=1131.001,321.659,-78.090,-177.656,10.657,149.522
C06172=1130.997,321.873,-78.118,-177.653,10.660,149.522
C06173=1130.994,322.085,-78.146,-177.651,10.662,149.522
C06174=1130.991,322.298,-78.175,-177.648,10.663,149.522
C06175=1130.986,322.546,-78.208,-177.645,10.666,149.522
C06176=1130.983,322.794,-78.242,-177.642,10.668,149.521
C06177=1130.979,323.042,-78.275,-177.639,10.671,149.521
C06178=1130.975,323.290,-78.308,-177.636,10.674,149.521
C06179=1130.971,323.537,-78.341,-177.632,10.676,149.521
C06180=1130.966,323.785,-78.374,-177.629,10.679,149.521
C06181=1130.962,324.033,-78.408,-177.626,10.681,149.521
C06182=1130.958,324.281,-78.441,-177.623,10.684,149.520
C06183=1130.954,324.528,-78.474,-177.619,10.686,149.520
C06184=1130.950,324.777,-78.507,-177.616,10.689,149.520
C06185=1130.947,325.024,-78.541,-177.613,10.691,149.520
C06186=1130.942,325.272,-78.574,-177.610,10.694,149.520
C06187=1130.938,325.519,-78.608,-177.607,10.697,149.520
C06188=1130.934,325.767,-78.641,-177.604,10.699,149.519
C06189=1130.930,326.015,-78.674,-177.600,10.702,149.519
C06190=1130.927,326.263,-78.708,-177.597,10.704,149.519
C06191=1130.923,326.510,-78.741,-177.594,10.707,149.519
C06192=1130.919,326.758,-78.775,-177.591,10.709,149.518
C06193=1130.914,327.006,-78.808,-177.587,10.712,149.518
C06194=1130.911,327.253,-78.842,-177.584,10.714,149.518
C06195=1130.906,327.501,-78.875,-177.581,10.717,149.518
C06196=1130.902,327.749,-78.909,-177.578,10.719,149.518
C06197=1130.898,327.996,-78.943,-177.575,10.721,149.518
C06198=1130.894,328.244,-78.976,-177.572,10.724,149.517
C06199=1130.890,328.492,-79.009,-177.569,10.726,149.517
C06200=1130.887,328.740,-79.043,-177.566,10.729,149.517
C06201=1130.883,328.987,-79.076,-177.563,10.731,149.517
C06202=1130.878,329.235,-79.111,-177.559,10.734,149.517
C06203=1130.874,329.483,-79.144,-177.556,10.736,149.516
C06204=1130.870,329.730,-79.177,-177.553,10.739,149.516
C06205=1130.867,329.978,-79.211,-177.550,10.742,149.516
C06206=1130.862,330.226,-79.245,-177.546,10.744,149.516
C06207=1130.858,330.473,-79.279,-177.543,10.746,149.515
C06208=1130.854,330.722,-79.313,-177.540,10.749,149.515
C06209=1130.851,330.969,-79.346,-177.537,10.752,149.515
C06210=1130.846,331.217,-79.380,-177.534,10.754,149.515
C06211=1130.842,331.464,-79.414,-177.530,10.757,149.515
C06212=1130.838,331.712,-79.448,-177.527,10.759,149.515
C06213=1130.834,331.959,-79.481,-177.524,10.762,149.514
C06214=1130.831,332.207,-79.515,-177.521,10.764,149.514
C06215=1130.826,332.455,-79.549,-177.517,10.767,149.514
C06216=1130.823,332.702,-79.583,-177.514,10.769,149.514
C06217=1130.818,332.950,-79.616,-177.511,10.772,149.514
C06218=1130.814,333.198,-79.651,-177.508,10.774,149.513
C06219=1130.811,333.445,-79.685,-177.504,10.777,149.513
C06220=1130.806,333.693,-79.718,-177.501,10.780,149.513
C06221=1130.802,333.941,-79.753,-177.499,10.781,149.513
C06222=1130.799,334.188,-79.787,-177.495,10.784,149.513
C06223=1130.795,334.401,-79.816,-177.493,10.787,149.513
C06224=1130.792,334.615,-79.845,-177.490,10.788,149.512
C06225=1130.788,334.828,-79.875,-177.487,10.791,149.512
C06226=1130.785,335.040,-79.904,-177.484,10.793,149.512
C06227=1130.782,335.254,-79.933,-177.482,10.795,149.512
C06228=1130.778,335.467,-79.962,-177.479,10.797,149.512
C06229=1130.775,335.681,-79.992,-177.476,10.799,149.511
C06230=1130.771,335.894,-80.021,-177.473,10.802,149.511
C06231=1130.767,336.141,-80.055,-177.470,10.804,149.511
C06232=1130.763,336.389,-80.090,-177.466,10.806,149.511
C06233=1130.759,336.636,-80.124,-177.463,10.809,149.511
C06234=1130.756,336.884,-80.158,-177.460,10.812,149.510
C06235=1130.752,337.131,-80.192,-177.457,10.814,149.510
C06236=1130.748,337.379,-80.226,-177.454,10.817,149.510
C06237=1130.744,337.627,-80.260,-177.451,10.819,149.510
C06238=1130.740,337.874,-80.294,-177.448,10.821,149.510
C06239=1130.736,338.122,-80.329,-177.445,10.824,149.509
C06240=1130.732,338.369,-80.363,-177.441,10.826,149.509
C06241=1130.728,338.617,-80.398,-177.438,10.828,149.509
C06242=1130.724,338.865,-80.432,-177.435,10.831,149.509
C06243=1130.720,339.112,-80.466,-177.432,10.834,149.509
C06244=1130.716,339.360,-80.500,-177.428,10.836,149.508
C06245=1130.712,339.607,-80.535,-177.425,10.839,149.508
C06246=1130.708,339.855,-80.570,-177.422,10.841,149.508
C06247=1130.704,340.102,-80.604,-177.419,10.844,149.508
C06248=1130.700,340.351,-80.638,-177.416,10.846,149.508
C06249=1130.696,340.598,-80.672,-177.412,10.849,149.507
C06250=1130.692,340.846,-80.707,-177.409,10.851,149.507
C06251=1130.688,341.093,-80.742,-177.406,10.854,149.507
C06252=1130.685,341.340,-80.776,-177.402,10.856,149.507
C06253=1130.680,341.588,-80.811,-177.399,10.859,149.507
C06254=1130.677,341.836,-80.845,-177.396,10.861,149.506
C06255=1130.672,342.083,-80.880,-177.393,10.864,149.506
C06256=1130.668,342.331,-80.914,-177.389,10.866,149.506
C06257=1130.665,342.578,-80.948,-177.386,10.869,149.506
C06258=1130.661,342.826,-80.984,-177.383,10.871,149.506
C06259=1130.656,343.073,-81.018,-177.380,10.874,149.505
C06260=1130.653,343.321,-81.053,-177.377,10.876,149.505
C06261=1130.648,343.568,-81.087,-177.373,10.879,149.505
C06262=1130.645,343.817,-81.122,-177.370,10.881,149.505
C06263=1130.640,344.063,-81.157,-177.367,10.884,149.505
C06264=1130.637,344.311,-81.191,-177.363,10.886,149.504
C06265=1130.632,344.559,-81.226,-177.360,10.889,149.504
C06266=1130.629,344.806,-81.261,-177.358,10.891,149.504
C06267=1130.625,345.054,-81.296,-177.354,10.893,149.504
C06268=1130.621,345.301,-81.330,-177.351,10.896,149.504
C06269=1130.617,345.549,-81.366,-177.348,10.898,149.503
C06270=1130.613,345.796,-81.400,-177.344,10.900,149.503
C06271=1130.609,346.044,-81.435,-177.341,10.903,149.503
C06272=1130.606,346.291,-81.470,-177.338,10.906,149.503
C06273=1130.601,346.539,-81.504,-177.335,10.908,149.503
C06274=1130.598,346.786,-81.540,-177.332,10.911,149.502
C06275=1130.593,347.034,-81.574,-177.328,10.913,149.502
C06276=1130.589,347.281,-81.610,-177.325,10.916,149.502
C06277=1130.586,347.529,-81.644,-177.322,10.918,149.502
C06278=1130.582,347.776,-81.679,-177.318,10.920,149.501
C06279=1130.578,347.990,-81.709,-177.315,10.923,149.501
C06280=1130.575,348.203,-81.740,-177.313,10.925,149.501
C06281=1130.572,348.415,-81.769,-177.310,10.927,149.501
C06282=1130.568,348.629,-81.800,-177.307,10.929,149.501
C06283=1130.564,348.841,-81.830,-177.304,10.931,149.501
C06284=1130.562,349.054,-81.860,-177.302,10.934,149.501
C06285=1130.558,349.267,-81.891,-177.299,10.936,149.500
C06286=1130.554,349.480,-81.921,-177.296,10.937,149.500
C06287=1130.550,349.728,-81.956,-177.292,10.940,149.500
C06288=1130.548,349.975,-81.991,-177.289,10.943,149.500
C06289=1130.543,350.222,-82.026,-177.285,10.946,149.499
C06290=1130.539,350.470,-82.061,-177.281,10.948,149.499
C06291=1130.536,350.718,-82.096,-177.277,10.952,149.499
C06292=1130.531,350.965,-82.131,-177.274,10.954,149.499
C06293=1130.527,351.213,-82.166,-177.271,10.956,149.498
C06294=1130.524,351.460,-82.202,-177.266,10.959,149.498
C06295=1130.520,351.708,-82.237,-177.263,10.962,149.498
C06296=1130.516,351.954,-82.272,-177.260,10.964,149.497
C06297=1130.512,352.203,-82.307,-177.256,10.968,149.497
C06298=1130.508,352.450,-82.343,-177.252,10.970,149.497
C06299=1130.505,352.698,-82.378,-177.249,10.972,149.497
C06300=1130.500,352.944,-82.413,-177.245,10.975,149.496
C06301=1130.497,353.192,-82.449,-177.241,10.978,149.496
C06302=1130.493,353.440,-82.484,-177.238,10.980,149.496
C06303=1130.489,353.688,-82.519,-177.234,10.983,149.496
C06304=1130.485,353.934,-82.555,-177.231,10.986,149.495
C06305=1130.481,354.182,-82.590,-177.227,10.988,149.495
C06306=1130.477,354.430,-82.626,-177.224,10.990,149.495
C06307=1130.473,354.677,-82.662,-177.220,10.994,149.495
C06308=1130.469,354.925,-82.697,-177.216,10.996,149.494
C06309=1130.466,355.172,-82.733,-177.213,10.998,149.494
C06310=1130.461,355.419,-82.768,-177.209,11.001,149.494
C06311=1130.458,355.666,-82.804,-177.205,11.004,149.494
C06312=1130.454,355.914,-82.839,-177.202,11.006,149.493
C06313=1130.450,356.161,-82.875,-177.198,11.008,149.493
C06314=1130.446,356.409,-82.911,-177.195,11.011,149.493
C06315=1130.442,356.657,-82.946,-177.191,11.013,149.492
C06316=1130.438,356.904,-82.982,-177.188,11.015,149.492
C06317=1130.434,357.151,-83.017,-177.184,11.019,149.492
C06318=1130.431,357.399,-83.053,-177.181,11.021,149.492
C06319=1130.427,357.646,-83.088,-177.177,11.023,149.491
C06320=1130.423,357.894,-83.124,-177.174,11.026,149.491
C06321=1130.419,358.141,-83.161,-177.170,11.028,149.491
C06322=1130.416,358.388,-83.196,-177.167,11.031,149.491
C06323=1130.412,358.636,-83.232,-177.163,11.033,149.490
C06324=1130.408,358.884,-83.268,-177.160,11.035,149.490
C06325=1130.404,359.131,-83.303,-177.156,11.039,149.490
C06326=1130.400,359.377,-83.339,-177.153,11.041,149.489
C06327=1130.396,359.625,-83.375,-177.149,11.043,149.489
C06328=1130.392,359.873,-83.411,-177.146,11.046,149.489
C06329=1130.388,360.120,-83.447,-177.143,11.048,149.489
C06330=1130.385,360.367,-83.483,-177.139,11.050,149.488
C06331=1130.381,360.615,-83.519,-177.136,11.053,149.488
C06332=1130.377,360.862,-83.555,-177.132,11.055,149.488
C06333=1130.374,361.109,-83.591,-177.129,11.058,149.488
C06334=1130.369,361.357,-83.627,-177.126,11.060,149.487
C06335=1130.366,361.570,-83.658,-177.123,11.062,149.487
C06336=1130.363,361.783,-83.689,-177.120,11.064,149.487
C06337=1130.360,361.996,-83.720,-177.117,11.066,149.487
C06338=1130.357,362.208,-83.751,-177.114,11.068,149.487
C06339=1130.353,362.421,-83.782,-177.111,11.070,149.486
C06340=1130.350,362.633,-83.813,-177.108,11.072,149.486
C06341=1130.347,362.846,-83.844,-177.105,11.074,149.486
C06342=1130.343,363.059,-83.875,-177.102,11.076,149.486
C06343=1130.340,363.306,-83.911,-177.099,11.078,149.485
C06344=1130.335,363.554,-83.947,-177.096,11.081,149.485
C06345=1130.332,363.801,-83.983,-177.092,11.083,149.485
C06346=1130.328,364.049,-84.019,-177.089,11.086,149.485
C06347=1130.324,364.296,-84.056,-177.085,11.088,149.484
C06348=1130.320,364.543,-84.092,-177.082,11.090,149.484
C06349=1130.317,364.790,-84.128,-177.079,11.093,149.484
C06350=1130.313,365.038,-84.164,-177.076,11.095,149.484
C06351=1130.309,365.285,-84.201,-177.073,11.097,149.483
C06352=1130.305,365.532,-84.237,-177.070,11.100,149.483
C06353=1130.301,365.780,-84.273,-177.066,11.102,149.483
C06354=1130.298,366.027,-84.310,-177.063,11.104,149.483
C06355=1130.294,366.275,-84.346,-177.059,11.107,149.482
C06356=1130.290,366.522,-84.383,-177.056,11.109,149.482
C06357=1130.286,366.769,-84.419,-177.053,11.112,149.482
C06358=1130.282,367.017,-84.455,-177.050,11.113,149.482
C06359=1130.279,367.264,-84.491,-177.047,11.116,149.481
C06360=1130.275,367.511,-84.528,-177.043,11.118,149.481
C06361=1130.271,367.758,-84.564,-177.040,11.121,149.481
C06362=1130.267,368.006,-84.601,-177.037,11.123,149.481
C06363=1130.263,368.253,-84.637,-177.033,11.126,149.481
C06364=1130.259,368.500,-84.674,-177.031,11.127,149.480
C06365=1130.256,368.748,-84.711,-177.027,11.130,149.480
C06366=1130.252,368.995,-84.746,-177.024,11.132,149.480
C06367=1130.248,369.242,-84.783,-177.021,11.135,149.480
C06368=1130.244,369.490,-84.820,-177.018,11.137,149.480
C06369=1130.241,369.736,-84.856,-177.015,11.139,149.479
C06370=1130.237,369.984,-84.893,-177.012,11.141,149.479
C06371=1130.233,370.231,-84.930,-177.008,11.144,149.479
C06372=1130.230,370.478,-84.967,-177.006,11.146,149.479
C06373=1130.225,370.726,-85.003,-177.002,11.148,149.478
C06374=1130.221,370.973,-85.040,-176.999,11.151,149.478
C06375=1130.218,371.220,-85.076,-176.996,11.153,149.478
C06376=1130.214,371.467,-85.113,-176.993,11.155,149.478
C06377=1130.210,371.715,-85.150,-176.990,11.157,149.478
C06378=1130.207,371.962,-85.186,-176.987,11.160,149.478
C06379=1130.203,372.209,-85.223,-176.984,11.162,149.477
C06380=1130.199,372.457,-85.260,-176.981,11.164,149.477
C06381=1130.195,372.704,-85.297,-176.978,11.167,149.477
C06382=1130.191,372.951,-85.333,-176.974,11.169,149.477
C06383=1130.188,373.199,-85.370,-176.972,11.171,149.476
C06384=1130.184,373.446,-85.407,-176.969,11.174,149.476
C06385=1130.180,373.693,-85.444,-176.965,11.176,149.476
C06386=1130.176,373.940,-85.480,-176.963,11.178,149.476
C06387=1130.173,374.188,-85.518,-176.959,11.180,149.476
C06388=1130.169,374.435,-85.554,-176.957,11.183,149.476
C06389=1130.165,374.681,-85.592,-176.954,11.185,149.475
C06390=1130.161,374.929,-85.629,-176.951,11.187,149.475
C06391=1130.158,375.141,-85.660,-176.948,11.189,149.475
C06392=1130.155,375.354,-85.691,-176.946,11.191,149.475
C06393=1130.152,375.567,-85.724,-176.943,11.193,149.475
C06394=1130.149,375.780,-85.756,-176.941,11.195,149.475
C06395=1130.145,375.993,-85.788,-176.938,11.197,149.475
C06396=1130.142,376.205,-85.820,-176.936,11.200,149.475
C06397=1130.138,376.418,-85.851,-176.933,11.201,149.474
C06398=1130.135,376.630,-85.883,-176.931,11.203,149.474
C06399=1130.132,376.877,-85.920,-176.928,11.205,149.474
C06400=1130.128,377.124,-85.957,-176.925,11.208,149.474
C06401=1130.124,377.372,-85.994,-176.922,11.210,149.474
C06402=1130.120,377.619,-86.031,-176.919,11.212,149.474
C06403=1130.116,377.866,-86.069,-176.916,11.215,149.474
C06404=1130.113,378.114,-86.106,-176.914,11.217,149.474
C06405=1130.109,378.361,-86.143,-176.911,11.219,149.473
C06406=1130.105,378.607,-86.180,-176.908,11.221,149.473
C06407=1130.102,378.855,-86.217,-176.905,11.224,149.473
C06408=1130.098,379.102,-86.254,-176.902,11.227,149.473
C06409=1130.094,379.349,-86.292,-176.899,11.228,149.473
C06410=1130.091,379.597,-86.329,-176.897,11.231,149.473
C06411=1130.087,379.844,-86.366,-176.894,11.233,149.473
C06412=1130.083,380.090,-86.403,-176.891,11.236,149.473
C06413=1130.079,380.338,-86.440,-176.889,11.238,149.472
C06414=1130.076,380.585,-86.478,-176.885,11.240,149.472
C06415=1130.071,380.832,-86.515,-176.883,11.242,149.472
C06416=1130.068,381.079,-86.553,-176.880,11.245,149.472
C06417=1130.064,381.326,-86.590,-176.878,11.247,149.472
C06418=1130.060,381.573,-86.627,-176.875,11.250,149.472
C06419=1130.057,381.821,-86.664,-176.872,11.252,149.472
C06420=1130.053,382.067,-86.702,-176.870,11.254,149.472
C06421=1130.050,382.315,-86.739,-176.867,11.257,149.472
C06422=1130.045,382.562,-86.777,-176.864,11.259,149.472
C06423=1130.041,382.809,-86.814,-176.861,11.262,149.472
C06424=1130.038,383.057,-86.852,-176.859,11.264,149.472
C06425=1130.034,383.304,-86.889,-176.856,11.267,149.472
C06426=1130.030,383.551,-86.927,-176.855,11.268,149.472
C06427=1130.026,383.798,-86.964,-176.853,11.270,149.472
C06428=1130.023,384.045,-87.001,-176.852,11.272,149.472
C06429=1130.019,384.292,-87.039,-176.850,11.274,149.472
C06430=1130.015,384.539,-87.076,-176.849,11.275,149.472
C06431=1130.012,384.787,-87.114,-176.848,11.277,149.472
C06432=1130.008,385.034,-87.151,-176.847,11.278,149.472
C06433=1130.005,385.281,-87.189,-176.845,11.280,149.472
C06434=1130.000,385.528,-87.227,-176.843,11.282,149.472
C06435=1129.996,385.775,-87.264,-176.842,11.284,149.473
C06436=1129.993,386.022,-87.302,-176.841,11.286,149.473
C06437=1129.989,386.269,-87.339,-176.840,11.287,149.473
C06438=1129.986,386.517,-87.377,-176.839,11.289,149.473
C06439=1129.982,386.764,-87.414,-176.837,11.292,149.473
C06440=1129.979,387.011,-87.452,-176.836,11.293,149.473
C06441=1129.974,387.258,-87.490,-176.835,11.295,149.474
C06442=1129.971,387.506,-87.528,-176.834,11.297,149.474
C06443=1129.967,387.752,-87.565,-176.833,11.299,149.474
C06444=1129.963,388.000,-87.602,-176.832,11.301,149.474
C06445=1129.960,388.247,-87.640,-176.830,11.303,149.474
C06446=1129.957,388.494,-87.678,-176.829,11.305,149.475
C06447=1129.953,388.706,-87.711,-176.829,11.307,149.475
C06448=1129.950,388.919,-87.743,-176.828,11.308,149.475
C06449=1129.947,389.131,-87.774,-176.827,11.310,149.475
C06450=1129.943,389.344,-87.807,-176.826,11.312,149.476
C06451=1129.940,389.557,-87.840,-176.825,11.313,149.476
C06452=1129.937,389.769,-87.873,-176.825,11.315,149.476
C06453=1129.934,389.981,-87.904,-176.824,11.317,149.476
C06454=1129.930,390.193,-87.937,-176.823,11.319,149.477
C06455=1129.927,390.441,-87.974,-176.822,11.321,149.477
C06456=1129.923,390.688,-88.012,-176.821,11.323,149.477
C06457=1129.919,390.935,-88.050,-176.820,11.325,149.478
C06458=1129.915,391.182,-88.088,-176.819,11.327,149.478
C06459=1129.912,391.429,-88.126,-176.818,11.329,149.478
C06460=1129.908,391.676,-88.163,-176.817,11.332,149.479
C06461=1129.905,391.924,-88.201,-176.816,11.334,149.479
C06462=1129.900,392.171,-88.239,-176.816,11.336,149.479
C06463=1129.897,392.418,-88.277,-176.815,11.338,149.480
C06464=1129.894,392.664,-88.314,-176.814,11.341,149.480
C06465=1129.890,392.912,-88.352,-176.813,11.343,149.481
C06466=1129.885,393.159,-88.390,-176.812,11.345,149.481
C06467=1129.882,393.406,-88.428,-176.811,11.348,149.481
C06468=1129.879,393.653,-88.465,-176.811,11.350,149.482
C06469=1129.875,393.900,-88.503,-176.810,11.353,149.482
C06470=1129.871,394.147,-88.541,-176.809,11.355,149.483
C06471=1129.868,394.394,-88.579,-176.808,11.358,149.483
C06472=1129.864,394.642,-88.617,-176.808,11.360,149.484
C06473=1129.860,394.889,-88.655,-176.807,11.362,149.484
C06474=1129.857,395.136,-88.693,-176.806,11.365,149.485
C06475=1129.853,395.383,-88.730,-176.806,11.367,149.485
C06476=1129.849,395.630,-88.768,-176.806,11.370,149.486
C06477=1129.845,395.877,-88.806,-176.805,11.373,149.486
C06478=1129.842,396.124,-88.844,-176.804,11.375,149.487
C06479=1129.838,396.371,-88.882,-176.804,11.378,149.487
C06480=1129.834,396.619,-88.920,-176.803,11.381,149.488
C06481=1129.830,396.865,-88.958,-176.803,11.383,149.488
C06482=1129.827,397.112,-88.996,-176.802,11.386,149.489
C06483=1129.823,397.359,-89.034,-176.801,11.389,149.489
C06484=1129.819,397.607,-89.072,-176.801,11.391,149.490
C06485=1129.816,397.854,-89.110,-176.801,11.394,149.491
C06486=1129.812,398.100,-89.148,-176.801,11.397,149.491
C06487=1129.808,398.348,-89.186,-176.800,11.400,149.492
C06488=1129.805,398.595,-89.224,-176.799,11.403,149.492
C06489=1129.801,398.842,-89.262,-176.799,11.405,149.493
C06490=1129.797,399.089,-89.300,-176.799,11.408,149.494
C06491=1129.794,399.336,-89.338,-176.799,11.411,149.494
C06492=1129.790,399.583,-89.375,-176.798,11.414,149.495
C06493=1129.786,399.830,-89.414,-176.798,11.417,149.496
C06494=1129.783,400.077,-89.452,-176.797,11.420,149.496
C06495=1129.778,400.324,-89.490,-176.797,11.423,149.497
C06496=1129.775,400.572,-89.528,-176.797,11.426,149.498
C06497=1129.771,400.818,-89.565,-176.797,11.429,149.499
C06498=1129.767,401.066,-89.604,-176.797,11.432,149.499
C06499=1129.764,401.313,-89.642,-176.796,11.435,149.500
C06500=1129.760,401.560,-89.679,-176.797,11.438,149.501
C06501=1129.756,401.807,-89.718,-176.796,11.442,149.502
C06502=1129.753,402.054,-89.756,-176.796,11.444,149.503
C06503=1129.750,402.266,-89.789,-176.796,11.447,149.503
C06504=1129.747,402.478,-89.822,-176.796,11.451,149.504
C06505=1129.743,402.691,-89.854,-176.796,11.453,149.505
C06506=1129.740,402.903,-89.887,-176.796,11.456,149.505
C06507=1129.737,403.116,-89.920,-176.796,11.459,149.506
C06508=1129.734,403.328,-89.952,-176.796,11.461,149.507
C06509=1129.731,403.540,-89.985,-176.796,11.465,149.508
C06510=1129.728,403.753,-90.018,-176.796,11.467,149.508
C06511=1129.724,404.000,-90.056,-176.796,11.470,149.509
C06512=1129.720,404.247,-90.094,-176.796,11.474,149.510
C06513=1129.717,404.494,-90.132,-176.796,11.477,149.511
C06514=1129.713,404.741,-90.170,-176.796,11.481,149.512
C06515=1129.709,404.989,-90.208,-176.796,11.485,149.513
C06516=1129.705,405.235,-90.247,-176.796,11.488,149.514
C06517=1129.702,405.482,-90.285,-176.796,11.492,149.515
C06518=1129.698,405.730,-90.324,-176.796,11.495,149.516
C06519=1129.694,405.976,-90.361,-176.797,11.499,149.517
C06520=1129.691,406.224,-90.399,-176.797,11.503,149.518
C06521=1129.687,406.471,-90.438,-176.798,11.506,149.519
C06522=1129.684,406.717,-90.476,-176.798,11.510,149.520
C06523=1129.680,406.965,-90.515,-176.798,11.514,149.521
C06524=1129.677,407.212,-90.553,-176.798,11.517,149.522
C06525=1129.672,407.459,-90.591,-176.799,11.521,149.523
C06526=1129.669,407.705,-90.629,-176.799,11.525,149.524
C06527=1129.665,407.952,-90.668,-176.799,11.529,149.525
C06528=1129.661,408.200,-90.705,-176.799,11.532,149.526
C06529=1129.658,408.447,-90.743,-176.800,11.536,149.527
C06530=1129.654,408.694,-90.782,-176.800,11.540,149.528
C06531=1129.651,408.940,-90.820,-176.801,11.544,149.530
C06532=1129.647,409.188,-90.859,-176.801,11.548,149.531
C06533=1129.643,409.435,-90.896,-176.802,11.552,149.532
C06534=1129.639,409.682,-90.935,-176.802,11.556,149.533
C06535=1129.636,409.929,-90.974,-176.802,11.561,149.534
C06536=1129.632,410.176,-91.012,-176.803,11.564,149.535
C06537=1129.629,410.423,-91.050,-176.804,11.568,149.537
C06538=1129.625,410.670,-91.089,-176.804,11.573,149.538
C06539=1129.621,410.916,-91.126,-176.805,11.577,149.539
C06540=1129.617,411.164,-91.165,-176.805,11.581,149.540
C06541=1129.614,411.411,-91.203,-176.806,11.585,149.542
C06542=1129.610,411.658,-91.242,-176.807,11.590,149.543
C06543=1129.607,411.905,-91.280,-176.807,11.594,149.544
C06544=1129.603,412.152,-91.318,-176.808,11.598,149.546
C06545=1129.599,412.398,-91.357,-176.809,11.603,149.547
C06546=1129.595,412.646,-91.395,-176.810,11.608,149.548
C06547=1129.592,412.893,-91.433,-176.810,11.612,149.550
C06548=1129.589,413.140,-91.472,-176.811,11.617,149.551
C06549=1129.585,413.387,-91.510,-176.812,11.620,149.552
C06550=1129.581,413.634,-91.548,-176.813,11.625,149.554
C06551=1129.577,413.881,-91.588,-176.814,11.630,149.555
C06552=1129.573,414.128,-91.625,-176.815,11.634,149.557
C06553=1129.571,414.375,-91.664,-176.816,11.639,149.558
C06554=1129.568,414.623,-91.702,-176.816,11.644,149.560
C06555=1129.566,414.870,-91.741,-176.817,11.648,149.561
C06556=1129.566,415.116,-91.778,-176.818,11.653,149.562
C06557=1129.565,415.363,-91.816,-176.819,11.658,149.564
C06558=1129.565,415.610,-91.855,-176.820,11.663,149.565
C06559=1129.565,415.823,-91.887,-176.821,11.667,149.567
C06560=1129.566,416.036,-91.919,-176.822,11.671,149.568
C06561=1129.567,416.247,-91.952,-176.823,11.675,149.569
C06562=1129.569,416.459,-91.984,-176.824,11.679,149.571
C06563=1129.572,416.672,-92.016,-176.825,11.684,149.572
C06564=1129.573,416.884,-92.048,-176.827,11.688,149.574
C06565=1129.577,417.097,-92.081,-176.827,11.692,149.575
C06566=1129.581,417.309,-92.113,-176.829,11.696,149.576
C06567=1129.161,417.308,-92.175,-176.821,11.701,149.576
C06568=1129.157,417.096,-92.143,-176.820,11.697,149.574
C06569=1129.154,416.884,-92.111,-176.819,11.692,149.573
C06570=1129.152,416.671,-92.079,-176.818,11.688,149.571
C06571=1129.150,416.459,-92.047,-176.817,11.684,149.570
C06572=1129.148,416.247,-92.014,-176.816,11.680,149.569
C06573=1129.146,416.035,-91.982,-176.815,11.675,149.567
C06574=1129.146,415.823,-91.950,-176.814,11.671,149.566
C06575=1129.146,415.610,-91.917,-176.813,11.667,149.565
C06576=1129.146,415.363,-91.879,-176.812,11.662,149.563
C06577=1129.146,415.116,-91.841,-176.811,11.658,149.562
C06578=1129.147,414.869,-91.803,-176.810,11.653,149.560
C06579=1129.148,414.622,-91.765,-176.809,11.648,149.559
C06580=1129.151,414.375,-91.726,-176.808,11.643,149.557
C06581=1129.155,414.128,-91.688,-176.807,11.639,149.556
C06582=1129.157,413.881,-91.649,-176.807,11.634,149.554
C06583=1129.161,413.634,-91.611,-176.806,11.629,149.553
C06584=1129.165,413.387,-91.573,-176.805,11.625,149.552
C06585=1129.169,413.140,-91.534,-176.804,11.620,149.550
C06586=1129.173,412.893,-91.495,-176.804,11.616,149.549
C06587=1129.176,412.647,-91.457,-176.803,11.611,149.548
C06588=1129.180,412.399,-91.419,-176.802,11.607,149.546
C06589=1129.183,412.152,-91.381,-176.802,11.602,149.545
C06590=1129.187,411.905,-91.341,-176.801,11.598,149.544
C06591=1129.191,411.658,-91.304,-176.801,11.593,149.542
C06592=1129.195,411.411,-91.265,-176.800,11.589,149.541
C06593=1129.197,411.164,-91.227,-176.799,11.585,149.540
C06594=1129.202,410.917,-91.189,-176.799,11.580,149.539
C06595=1129.205,410.670,-91.151,-176.798,11.576,149.537
C06596=1129.209,410.422,-91.112,-176.798,11.572,149.536
C06597=1129.213,410.176,-91.074,-176.797,11.568,149.535
C06598=1129.217,409.929,-91.035,-176.797,11.564,149.534
C06599=1129.220,409.681,-90.997,-176.796,11.560,149.533
C06600=1129.224,409.435,-90.958,-176.796,11.555,149.531
C06601=1129.227,409.188,-90.920,-176.796,11.551,149.530
C06602=1129.231,408.940,-90.882,-176.795,11.547,149.529
C06603=1129.235,408.694,-90.844,-176.795,11.544,149.528
C06604=1129.238,408.447,-90.805,-176.794,11.540,149.527
C06605=1129.242,408.200,-90.767,-176.794,11.536,149.526
C06606=1129.246,407.953,-90.729,-176.794,11.532,149.525
C06607=1129.249,407.705,-90.691,-176.793,11.528,149.524
C06608=1129.253,407.458,-90.652,-176.793,11.524,149.523
C06609=1129.257,407.212,-90.614,-176.793,11.520,149.521
C06610=1129.261,406.964,-90.576,-176.793,11.516,149.520
C06611=1129.264,406.717,-90.538,-176.792,11.513,149.519
C06612=1129.267,406.471,-90.499,-176.792,11.509,149.518
C06613=1129.271,406.223,-90.461,-176.792,11.505,149.517
C06614=1129.274,405.976,-90.423,-176.792,11.501,149.516
C06615=1129.279,405.729,-90.385,-176.792,11.498,149.515
C06616=1129.282,405.482,-90.347,-176.792,11.494,149.514
C06617=1129.286,405.236,-90.308,-176.792,11.491,149.513
C06618=1129.290,404.989,-90.270,-176.791,11.487,149.512
C06619=1129.293,404.741,-90.232,-176.792,11.484,149.512
C06620=1129.297,404.494,-90.194,-176.792,11.480,149.511
C06621=1129.300,404.247,-90.156,-176.791,11.477,149.510
C06622=1129.304,403.999,-90.117,-176.792,11.473,149.509
C06623=1129.308,403.754,-90.079,-176.791,11.470,149.508
C06624=1129.311,403.541,-90.046,-176.792,11.467,149.507
C06625=1129.314,403.328,-90.014,-176.792,11.464,149.506
C06626=1129.318,403.116,-89.981,-176.791,11.461,149.506
C06627=1129.321,402.903,-89.948,-176.791,11.459,149.505
C06628=1129.324,402.691,-89.915,-176.792,11.455,149.504
C06629=1129.327,402.479,-89.882,-176.792,11.452,149.503
C06630=1129.330,402.267,-89.850,-176.792,11.450,149.503
C06631=1129.333,402.054,-89.817,-176.792,11.447,149.502
C06632=1129.337,401.807,-89.779,-176.792,11.444,149.501
C06633=1129.341,401.559,-89.741,-176.792,11.441,149.501
C06634=1129.345,401.313,-89.703,-176.793,11.437,149.500
C06635=1129.348,401.066,-89.664,-176.793,11.435,149.499
C06636=1129.352,400.819,-89.627,-176.793,11.431,149.498
C06637=1129.356,400.572,-89.588,-176.793,11.429,149.498
C06638=1129.359,400.325,-89.550,-176.794,11.425,149.497
C06639=1129.363,400.078,-89.513,-176.794,11.423,149.496
C06640=1129.367,399.830,-89.474,-176.794,11.419,149.495
C06641=1129.370,399.584,-89.437,-176.794,11.416,149.495
C06642=1129.374,399.337,-89.399,-176.795,11.413,149.494
C06643=1129.377,399.089,-89.360,-176.795,11.411,149.493
C06644=1129.381,398.842,-89.323,-176.796,11.407,149.493
C06645=1129.384,398.595,-89.285,-176.796,11.405,149.492
C06646=1129.389,398.348,-89.246,-176.797,11.402,149.492
C06647=1129.392,398.101,-89.209,-176.797,11.399,149.491
C06648=1129.396,397.854,-89.171,-176.798,11.396,149.490
C06649=1129.400,397.607,-89.132,-176.798,11.394,149.490
C06650=1129.403,397.360,-89.094,-176.799,11.390,149.489
C06651=1129.407,397.113,-89.057,-176.799,11.388,149.488
C06652=1129.411,396.865,-89.018,-176.799,11.385,149.488
C06653=1129.415,396.619,-88.981,-176.800,11.382,149.487
C06654=1129.418,396.372,-88.943,-176.801,11.380,149.487
C06655=1129.422,396.125,-88.905,-176.802,11.377,149.486
C06656=1129.425,395.877,-88.867,-176.802,11.375,149.486
C06657=1129.429,395.631,-88.829,-176.802,11.372,149.485
C06658=1129.433,395.383,-88.791,-176.803,11.369,149.485
C06659=1129.437,395.136,-88.754,-176.804,11.367,149.484
C06660=1129.440,394.889,-88.716,-176.805,11.364,149.484
C06661=1129.444,394.642,-88.678,-176.805,11.362,149.483
C06662=1129.448,394.395,-88.640,-176.806,11.359,149.483
C06663=1129.451,394.147,-88.602,-176.807,11.356,149.482
C06664=1129.455,393.901,-88.564,-176.807,11.354,149.482
C06665=1129.459,393.653,-88.526,-176.808,11.352,149.482
C06666=1129.463,393.407,-88.488,-176.809,11.349,149.481
C06667=1129.466,393.159,-88.450,-176.810,11.347,149.481
C06668=1129.470,392.912,-88.413,-176.811,11.345,149.480
C06669=1129.474,392.665,-88.375,-176.812,11.342,149.480
C06670=1129.478,392.418,-88.337,-176.812,11.340,149.480
C06671=1129.481,392.171,-88.299,-176.813,11.338,149.479
C06672=1129.485,391.924,-88.262,-176.814,11.335,149.479
C06673=1129.488,391.677,-88.224,-176.815,11.333,149.478
C06674=1129.493,391.429,-88.186,-176.816,11.331,149.478
C06675=1129.496,391.182,-88.148,-176.817,11.329,149.478
C06676=1129.500,390.936,-88.111,-176.818,11.326,149.477
C06677=1129.503,390.688,-88.073,-176.819,11.324,149.477
C06678=1129.507,390.442,-88.035,-176.819,11.322,149.477
C06679=1129.511,390.194,-87.997,-176.821,11.320,149.476
C06680=1129.514,389.982,-87.965,-176.822,11.318,149.476
C06681=1129.517,389.769,-87.933,-176.823,11.316,149.476
C06682=1129.521,389.557,-87.900,-176.823,11.315,149.476
C06683=1129.524,389.344,-87.867,-176.824,11.313,149.476
C06684=1129.526,389.132,-87.835,-176.825,11.311,149.475
C06685=1129.530,388.919,-87.803,-176.826,11.309,149.475
C06686=1129.533,388.707,-87.770,-176.827,11.307,149.475
C06687=1129.536,388.494,-87.739,-176.828,11.306,149.475
C06688=1129.540,388.247,-87.700,-176.829,11.304,149.474
C06689=1129.544,388.000,-87.663,-176.830,11.301,149.474
C06690=1129.547,387.753,-87.625,-176.831,11.300,149.474
C06691=1129.551,387.506,-87.588,-176.832,11.298,149.474
C06692=1129.555,387.259,-87.550,-176.834,11.296,149.474
C06693=1129.558,387.012,-87.512,-176.835,11.294,149.473
C06694=1129.563,386.764,-87.475,-176.836,11.292,149.473
C06695=1129.566,386.517,-87.437,-176.837,11.290,149.473
C06696=1129.570,386.270,-87.399,-176.838,11.289,149.473
C06697=1129.574,386.023,-87.362,-176.840,11.287,149.473
C06698=1129.577,385.776,-87.325,-176.841,11.284,149.472
C06699=1129.581,385.529,-87.287,-176.842,11.283,149.472
C06700=1129.585,385.282,-87.250,-176.844,11.281,149.472
C06701=1129.588,385.034,-87.212,-176.845,11.280,149.472
C06702=1129.592,384.788,-87.174,-176.847,11.277,149.472
C06703=1129.596,384.540,-87.137,-176.848,11.276,149.472
C06704=1129.600,384.293,-87.099,-176.849,11.274,149.472
C06705=1129.603,384.045,-87.062,-176.850,11.273,149.472
C06706=1129.607,383.799,-87.024,-176.852,11.271,149.472
C06707=1129.611,383.552,-86.987,-176.854,11.269,149.472
C06708=1129.614,383.304,-86.949,-176.855,11.267,149.471
C06709=1129.618,383.058,-86.912,-176.858,11.264,149.471
C06710=1129.622,382.810,-86.875,-176.860,11.262,149.472
C06711=1129.625,382.563,-86.837,-176.863,11.260,149.472
C06712=1129.629,382.316,-86.800,-176.866,11.258,149.472
C06713=1129.633,382.069,-86.762,-176.868,11.255,149.472
C06714=1129.637,381.821,-86.725,-176.871,11.253,149.472
C06715=1129.640,381.574,-86.687,-176.874,11.250,149.472
C06716=1129.644,381.327,-86.651,-176.876,11.248,149.472
C06717=1129.648,381.080,-86.613,-176.879,11.245,149.472
C06718=1129.651,380.833,-86.576,-176.882,11.243,149.472
C06719=1129.655,380.586,-86.538,-176.885,11.241,149.472
C06720=1129.659,380.339,-86.501,-176.888,11.238,149.472
C06721=1129.662,380.092,-86.463,-176.890,11.236,149.472
C06722=1129.666,379.844,-86.427,-176.893,11.234,149.473
C06723=1129.671,379.597,-86.390,-176.896,11.232,149.473
C06724=1129.674,379.350,-86.352,-176.899,11.229,149.473
C06725=1129.678,379.103,-86.315,-176.901,11.227,149.473
C06726=1129.682,378.856,-86.277,-176.904,11.224,149.473
C06727=1129.685,378.608,-86.240,-176.907,11.222,149.473
C06728=1129.689,378.361,-86.203,-176.910,11.220,149.473
C06729=1129.693,378.114,-86.166,-176.913,11.217,149.473
C06730=1129.696,377.867,-86.128,-176.915,11.215,149.473
C06731=1129.701,377.619,-86.092,-176.918,11.213,149.474
C06732=1129.705,377.372,-86.055,-176.921,11.210,149.474
C06733=1129.708,377.125,-86.017,-176.924,11.208,149.474
C06734=1129.712,376.878,-85.980,-176.927,11.206,149.474
C06735=1129.716,376.631,-85.943,-176.930,11.204,149.474
C06736=1129.719,376.418,-85.912,-176.933,11.201,149.474
C06737=1129.723,376.206,-85.879,-176.935,11.199,149.474
C06738=1129.726,375.993,-85.848,-176.937,11.197,149.474
C06739=1129.728,375.781,-85.816,-176.940,11.196,149.475
C06740=1129.732,375.568,-85.784,-176.942,11.194,149.475
C06741=1129.735,375.355,-85.752,-176.945,11.192,149.475
C06742=1129.738,375.142,-85.720,-176.947,11.190,149.475
C06743=1129.741,374.930,-85.689,-176.950,11.188,149.475
C06744=1129.745,374.682,-85.652,-176.953,11.185,149.475
C06745=1129.749,374.435,-85.615,-176.956,11.183,149.476
C06746=1129.753,374.188,-85.578,-176.959,11.181,149.476
C06747=1129.756,373.940,-85.541,-176.962,11.179,149.476
C06748=1129.760,373.693,-85.504,-176.965,11.176,149.476
C06749=1129.764,373.446,-85.468,-176.968,11.174,149.476
C06750=1129.768,373.199,-85.430,-176.971,11.172,149.476
C06751=1129.771,372.953,-85.394,-176.974,11.169,149.477
C06752=1129.775,372.705,-85.357,-176.977,11.167,149.477
C06753=1129.779,372.457,-85.320,-176.980,11.165,149.477
C06754=1129.783,372.210,-85.283,-176.983,11.162,149.477
C06755=1129.787,371.963,-85.247,-176.986,11.160,149.477
C06756=1129.790,371.715,-85.209,-176.989,11.158,149.478
C06757=1129.794,371.468,-85.172,-176.992,11.156,149.478
C06758=1129.798,371.221,-85.137,-176.996,11.153,149.478
C06759=1129.802,370.974,-85.100,-176.998,11.151,149.478
C06760=1129.806,370.726,-85.063,-177.002,11.149,149.478
C06761=1129.810,370.479,-85.026,-177.005,11.146,149.479
C06762=1129.813,370.232,-84.990,-177.008,11.144,149.479
C06763=1129.817,369.984,-84.953,-177.011,11.142,149.479
C06764=1129.821,369.737,-84.916,-177.014,11.139,149.479
C06765=1129.824,369.490,-84.880,-177.017,11.137,149.479
C06766=1129.829,369.243,-84.844,-177.020,11.134,149.480
C06767=1129.832,368.996,-84.807,-177.024,11.132,149.480
C06768=1129.836,368.749,-84.770,-177.026,11.130,149.480
C06769=1129.840,368.501,-84.733,-177.030,11.128,149.480
C06770=1129.843,368.254,-84.697,-177.033,11.125,149.480
C06771=1129.847,368.006,-84.661,-177.036,11.123,149.481
C06772=1129.851,367.759,-84.625,-177.040,11.121,149.481
C06773=1129.855,367.512,-84.588,-177.043,11.119,149.481
C06774=1129.859,367.265,-84.551,-177.046,11.117,149.482
C06775=1129.863,367.017,-84.515,-177.049,11.114,149.482
C06776=1129.867,366.770,-84.478,-177.053,11.112,149.482
C06777=1129.870,366.523,-84.442,-177.056,11.109,149.482
C06778=1129.875,366.275,-84.406,-177.059,11.107,149.482
C06779=1129.878,366.028,-84.370,-177.062,11.105,149.483
C06780=1129.881,365.781,-84.333,-177.065,11.103,149.483
C06781=1129.885,365.533,-84.297,-177.069,11.100,149.483
C06782=1129.889,365.286,-84.260,-177.072,11.098,149.483
C06783=1129.893,365.038,-84.225,-177.076,11.095,149.484
C06784=1129.897,364.791,-84.188,-177.079,11.093,149.484
C06785=1129.901,364.544,-84.152,-177.082,11.090,149.484
C06786=1129.905,364.296,-84.115,-177.085,11.088,149.484
C06787=1129.908,364.050,-84.079,-177.089,11.086,149.485
C06788=1129.912,363.802,-84.043,-177.091,11.084,149.485
C06789=1129.916,363.555,-84.007,-177.095,11.082,149.485
C06790=1129.919,363.307,-83.971,-177.098,11.079,149.485
C06791=1129.924,363.060,-83.935,-177.102,11.077,149.486
C06792=1129.927,362.847,-83.904,-177.105,11.074,149.486
C06793=1129.930,362.634,-83.872,-177.108,11.073,149.486
C06794=1129.933,362.422,-83.841,-177.110,11.071,149.486
C06795=1129.937,362.209,-83.811,-177.114,11.068,149.487
C06796=1129.940,361.996,-83.780,-177.116,11.066,149.487
C06797=1129.943,361.784,-83.748,-177.119,11.064,149.487
C06798=1129.946,361.570,-83.718,-177.122,11.062,149.487
C06799=1129.949,361.358,-83.687,-177.125,11.060,149.487
C06800=1129.954,361.110,-83.650,-177.129,11.057,149.488
C06801=1129.957,360.863,-83.614,-177.132,11.055,149.488
C06802=1129.961,360.616,-83.579,-177.136,11.053,149.488
C06803=1129.964,360.368,-83.543,-177.139,11.050,149.488
C06804=1129.969,360.120,-83.507,-177.142,11.048,149.489
C06805=1129.972,359.873,-83.471,-177.146,11.046,149.489
C06806=1129.976,359.627,-83.436,-177.149,11.043,149.489
C06807=1129.981,359.379,-83.399,-177.153,11.041,149.489
C06808=1129.985,359.131,-83.364,-177.156,11.038,149.490
C06809=1129.988,358.884,-83.328,-177.160,11.036,149.490
C06810=1129.992,358.637,-83.292,-177.163,11.034,149.490
C06811=1129.996,358.389,-83.256,-177.166,11.031,149.490
C06812=1130.000,358.142,-83.220,-177.169,11.029,149.491
C06813=1130.003,357.894,-83.185,-177.173,11.027,149.491
C06814=1130.007,357.647,-83.149,-177.177,11.023,149.491
C06815=1130.010,357.400,-83.113,-177.180,11.021,149.491
C06816=1130.015,357.152,-83.077,-177.184,11.019,149.492
C06817=1130.019,356.905,-83.042,-177.187,11.016,149.492
C06818=1130.023,356.658,-83.006,-177.191,11.014,149.492
C06819=1130.026,356.410,-82.971,-177.194,11.011,149.493
C06820=1130.030,356.163,-82.935,-177.198,11.009,149.493
C06821=1130.034,355.915,-82.899,-177.202,11.006,149.493
C06822=1130.038,355.667,-82.863,-177.205,11.004,149.493
C06823=1130.042,355.420,-82.828,-177.208,11.001,149.494
C06824=1130.046,355.173,-82.793,-177.212,10.999,149.494
C06825=1130.050,354.925,-82.757,-177.215,10.996,149.494
C06826=1130.053,354.678,-82.721,-177.219,10.993,149.494
C06827=1130.057,354.430,-82.686,-177.223,10.991,149.495
C06828=1130.061,354.183,-82.650,-177.226,10.989,149.495
C06829=1130.065,353.936,-82.615,-177.230,10.986,149.495
C06830=1130.069,353.689,-82.580,-177.233,10.983,149.495
C06831=1130.072,353.441,-82.544,-177.237,10.981,149.496
C06832=1130.077,353.193,-82.509,-177.241,10.978,149.496
C06833=1130.081,352.945,-82.473,-177.244,10.975,149.496
C06834=1130.085,352.698,-82.438,-177.248,10.973,149.497
C06835=1130.088,352.451,-82.402,-177.251,10.970,149.497
C06836=1130.092,352.203,-82.367,-177.255,10.967,149.497
C06837=1130.096,351.955,-82.332,-177.259,10.965,149.497
C06838=1130.100,351.709,-82.297,-177.262,10.963,149.498
C06839=1130.104,351.461,-82.261,-177.266,10.959,149.498
C06840=1130.108,351.214,-82.226,-177.270,10.957,149.498
C06841=1130.112,350.965,-82.191,-177.273,10.954,149.498
C06842=1130.116,350.719,-82.156,-177.277,10.952,149.499
C06843=1130.119,350.471,-82.121,-177.281,10.949,149.499
C06844=1130.123,350.223,-82.086,-177.285,10.946,149.499
C06845=1130.127,349.977,-82.051,-177.288,10.943,149.499
C06846=1130.131,349.729,-82.015,-177.292,10.941,149.500
C06847=1130.135,349.481,-81.980,-177.296,10.938,149.500
C06848=1130.139,349.268,-81.950,-177.298,10.936,149.500
C06849=1130.142,349.055,-81.920,-177.301,10.934,149.500
C06850=1130.145,348.842,-81.890,-177.304,10.932,149.501
C06851=1130.149,348.629,-81.859,-177.306,10.930,149.501
C06852=1130.151,348.417,-81.829,-177.309,10.927,149.501
C06853=1130.155,348.204,-81.799,-177.312,10.926,149.501
C06854=1130.159,347.991,-81.769,-177.315,10.923,149.501
C06855=1130.162,347.778,-81.739,-177.318,10.921,149.501
C06856=1130.166,347.530,-81.704,-177.321,10.919,149.502
C06857=1130.169,347.283,-81.669,-177.324,10.916,149.502
C06858=1130.174,347.035,-81.634,-177.327,10.914,149.502
C06859=1130.178,346.787,-81.599,-177.331,10.911,149.502
C06860=1130.181,346.540,-81.565,-177.334,10.909,149.502
C06861=1130.185,346.293,-81.530,-177.337,10.906,149.503
C06862=1130.189,346.045,-81.494,-177.341,10.904,149.503
C06863=1130.194,345.798,-81.460,-177.344,10.901,149.503
C06864=1130.198,345.550,-81.425,-177.347,10.899,149.503
C06865=1130.201,345.302,-81.390,-177.350,10.896,149.504
C06866=1130.205,345.055,-81.356,-177.353,10.894,149.504
C06867=1130.209,344.807,-81.320,-177.357,10.891,149.504
C06868=1130.213,344.560,-81.286,-177.360,10.889,149.504
C06869=1130.217,344.312,-81.252,-177.363,10.886,149.504
C06870=1130.221,344.065,-81.217,-177.367,10.884,149.505
C06871=1130.225,343.817,-81.182,-177.370,10.881,149.505
C06872=1130.229,343.569,-81.147,-177.373,10.878,149.505
C06873=1130.233,343.322,-81.113,-177.376,10.876,149.505
C06874=1130.237,343.074,-81.078,-177.379,10.874,149.505
C06875=1130.241,342.827,-81.043,-177.382,10.872,149.506
C06876=1130.244,342.579,-81.009,-177.385,10.869,149.506
C06877=1130.249,342.332,-80.974,-177.389,10.867,149.506
C06878=1130.253,342.084,-80.939,-177.392,10.864,149.506
C06879=1130.256,341.837,-80.905,-177.395,10.862,149.506
C06880=1130.260,341.589,-80.870,-177.398,10.859,149.507
C06881=1130.265,341.342,-80.835,-177.402,10.857,149.507
C06882=1130.268,341.094,-80.801,-177.405,10.854,149.507
C06883=1130.272,340.847,-80.767,-177.408,10.852,149.507
C06884=1130.276,340.599,-80.732,-177.411,10.849,149.507
C06885=1130.280,340.351,-80.698,-177.415,10.847,149.508
C06886=1130.284,340.103,-80.663,-177.418,10.844,149.508
C06887=1130.288,339.856,-80.629,-177.421,10.842,149.508
C06888=1130.292,339.608,-80.594,-177.424,10.839,149.508
C06889=1130.296,339.361,-80.561,-177.427,10.837,149.508
C06890=1130.300,339.113,-80.526,-177.431,10.834,149.509
C06891=1130.304,338.866,-80.492,-177.434,10.832,149.509
C06892=1130.308,338.618,-80.457,-177.437,10.829,149.509
C06893=1130.311,338.370,-80.423,-177.441,10.827,149.509
C06894=1130.316,338.123,-80.389,-177.444,10.824,149.509
C06895=1130.319,337.875,-80.354,-177.447,10.822,149.510
C06896=1130.324,337.628,-80.320,-177.450,10.819,149.510
C06897=1130.328,337.381,-80.286,-177.454,10.817,149.510
C06898=1130.332,337.133,-80.251,-177.457,10.814,149.510
C06899=1130.335,336.885,-80.217,-177.460,10.811,149.510
C06900=1130.340,336.637,-80.183,-177.463,10.809,149.511
C06901=1130.344,336.390,-80.149,-177.466,10.806,149.511
C06902=1130.348,336.141,-80.115,-177.469,10.805,149.511
C06903=1130.351,335.894,-80.081,-177.472,10.802,149.511
C06904=1130.355,335.681,-80.052,-177.475,10.800,149.511
C06905=1130.358,335.468,-80.023,-177.478,10.798,149.511
C06906=1130.362,335.255,-79.992,-177.481,10.795,149.512
C06907=1130.365,335.042,-79.964,-177.484,10.793,149.512
C06908=1130.368,334.829,-79.934,-177.486,10.791,149.512
C06909=1130.372,334.616,-79.905,-177.489,10.789,149.512
C06910=1130.376,334.403,-79.876,-177.492,10.787,149.512
C06911=1130.379,334.190,-79.846,-177.495,10.785,149.513
C06912=1130.383,333.942,-79.813,-177.498,10.782,149.513
C06913=1130.387,333.694,-79.778,-177.501,10.779,149.513
C06914=1130.391,333.447,-79.744,-177.504,10.777,149.513
C06915=1130.395,333.199,-79.711,-177.508,10.774,149.513
C06916=1130.398,332.951,-79.677,-177.511,10.772,149.513
C06917=1130.402,332.704,-79.642,-177.513,10.770,149.514
C06918=1130.407,332.456,-79.609,-177.517,10.767,149.514
C06919=1130.410,332.209,-79.575,-177.520,10.765,149.514
C06920=1130.415,331.960,-79.541,-177.523,10.762,149.514
C06921=1130.419,331.713,-79.507,-177.526,10.760,149.514
C06922=1130.422,331.466,-79.473,-177.530,10.757,149.515
C06923=1130.426,331.218,-79.440,-177.533,10.755,149.515
C06924=1130.431,330.970,-79.405,-177.536,10.752,149.515
C06925=1130.435,330.723,-79.372,-177.539,10.750,149.515
C06926=1130.438,330.475,-79.338,-177.542,10.747,149.516
C06927=1130.442,330.227,-79.305,-177.545,10.744,149.516
C06928=1130.447,329.980,-79.270,-177.549,10.742,149.516
C06929=1130.451,329.732,-79.237,-177.552,10.740,149.516
C06930=1130.454,329.483,-79.204,-177.555,10.737,149.516
C06931=1130.458,329.236,-79.170,-177.558,10.734,149.516
C06932=1130.462,328.989,-79.137,-177.562,10.732,149.517
C06933=1130.466,328.741,-79.103,-177.565,10.729,149.517
C06934=1130.471,328.493,-79.069,-177.568,10.727,149.517
C06935=1130.474,328.245,-79.035,-177.571,10.724,149.517
C06936=1130.478,327.998,-79.002,-177.574,10.722,149.517
C06937=1130.482,327.750,-78.968,-177.578,10.719,149.518
C06938=1130.487,327.502,-78.935,-177.581,10.717,149.518
C06939=1130.490,327.255,-78.901,-177.584,10.714,149.518
C06940=1130.494,327.007,-78.868,-177.587,10.712,149.518
C06941=1130.498,326.759,-78.835,-177.590,10.710,149.518
C06942=1130.503,326.512,-78.800,-177.593,10.707,149.519
C06943=1130.507,326.264,-78.767,-177.596,10.705,149.519
C06944=1130.511,326.016,-78.734,-177.600,10.702,149.519
C06945=1130.514,325.768,-78.700,-177.603,10.700,149.519
C06946=1130.518,325.521,-78.667,-177.606,10.697,149.519
C06947=1130.522,325.273,-78.633,-177.609,10.695,149.520
C06948=1130.527,325.025,-78.600,-177.612,10.692,149.520
C06949=1130.531,324.778,-78.567,-177.615,10.689,149.520
C06950=1130.535,324.530,-78.534,-177.619,10.687,149.520
C06951=1130.539,324.282,-78.501,-177.622,10.684,149.520
C06952=1130.542,324.034,-78.467,-177.625,10.682,149.520
C06953=1130.546,323.787,-78.433,-177.628,10.679,149.521
C06954=1130.551,323.539,-78.400,-177.631,10.677,149.521
C06955=1130.555,323.291,-78.367,-177.635,10.674,149.521
C06956=1130.559,323.043,-78.334,-177.638,10.672,149.521
C06957=1130.563,322.796,-78.301,-177.641,10.669,149.521
C06958=1130.567,322.548,-78.268,-177.644,10.666,149.522
C06959=1130.570,322.300,-78.235,-177.647,10.664,149.522
C06960=1130.573,322.087,-78.206,-177.650,10.662,149.522
C06961=1130.577,321.873,-78.178,-177.652,10.660,149.522
C06962=1130.581,321.661,-78.149,-177.655,10.658,149.522
C06963=1130.585,321.447,-78.121,-177.658,10.656,149.522
C06964=1130.588,321.234,-78.092,-177.661,10.653,149.523
C06965=1130.591,321.021,-78.064,-177.663,10.651,149.523
C06966=1130.595,320.808,-78.035,-177.666,10.649,149.523
C06967=1130.598,320.594,-78.007,-177.669,10.647,149.523
C06968=1130.602,320.346,-77.974,-177.672,10.644,149.523
C06969=1130.606,320.098,-77.940,-177.675,10.641,149.523
C06970=1130.610,319.851,-77.907,-177.678,10.639,149.524
C06971=1130.614,319.603,-77.875,-177.682,10.637,149.524
C06972=1130.618,319.355,-77.842,-177.685,10.634,149.524
C06973=1130.622,319.107,-77.809,-177.688,10.631,149.524
C06974=1130.626,318.859,-77.776,-177.691,10.630,149.525
C06975=1130.631,318.612,-77.743,-177.694,10.627,149.525
C06976=1130.634,318.364,-77.710,-177.697,10.625,149.525
C06977=1130.638,318.117,-77.677,-177.700,10.622,149.525
C06978=1130.643,317.868,-77.645,-177.703,10.619,149.525
C06979=1130.647,317.620,-77.611,-177.707,10.617,149.525
C06980=1130.650,317.373,-77.579,-177.710,10.614,149.525
C06981=1130.654,317.125,-77.546,-177.713,10.612,149.526
C06982=1130.659,316.877,-77.513,-177.716,10.609,149.526
C06983=1130.663,316.629,-77.480,-177.719,10.606,149.526
C06984=1130.666,316.382,-77.448,-177.722,10.604,149.526
C06985=1130.671,316.133,-77.415,-177.726,10.602,149.527
C06986=1130.675,315.886,-77.382,-177.729,10.599,149.527
C06987=1130.678,315.638,-77.349,-177.732,10.596,149.527
C06988=1130.683,315.390,-77.317,-177.735,10.594,149.527
C06989=1130.687,315.142,-77.284,-177.738,10.591,149.527
C06990=1130.690,314.895,-77.251,-177.742,10.589,149.527
C06991=1130.695,314.647,-77.219,-177.745,10.586,149.528
C06992=1130.699,314.399,-77.186,-177.748,10.583,149.528
C06993=1130.703,314.151,-77.154,-177.751,10.582,149.528
C06994=1130.707,313.904,-77.121,-177.753,10.579,149.528
C06995=1130.712,313.655,-77.089,-177.757,10.577,149.528
C06996=1130.715,313.408,-77.056,-177.760,10.574,149.528
C06997=1130.720,313.160,-77.024,-177.763,10.571,149.529
C06998=1130.723,312.912,-76.991,-177.766,10.569,149.529
C06999=1130.727,312.664,-76.959,-177.769,10.566,149.529
C07000=1130.731,312.416,-76.926,-177.773,10.564,149.529
C07001=1130.736,312.169,-76.894,-177.776,10.561,149.529
C07002=1130.740,311.921,-76.861,-177.779,10.559,149.530
C07003=1130.744,311.673,-76.829,-177.782,10.556,149.530
C07004=1130.748,311.425,-76.796,-177.785,10.553,149.530
C07005=1130.751,311.177,-76.764,-177.789,10.551,149.530
C07006=1130.756,310.929,-76.732,-177.791,10.548,149.530
C07007=1130.759,310.681,-76.699,-177.795,10.546,149.531
C07008=1130.764,310.434,-76.667,-177.798,10.543,149.531
C07009=1130.768,310.186,-76.635,-177.801,10.540,149.531
C07010=1130.772,309.938,-76.602,-177.804,10.539,149.531
C07011=1130.776,309.690,-76.570,-177.807,10.536,149.531
C07012=1130.780,309.442,-76.538,-177.810,10.534,149.532
C07013=1130.785,309.194,-76.506,-177.813,10.531,149.532
C07014=1130.789,308.947,-76.473,-177.816,10.528,149.532
C07015=1130.793,308.698,-76.441,-177.819,10.526,149.532
C07016=1130.796,308.485,-76.413,-177.823,10.523,149.532
C07017=1130.799,308.272,-76.385,-177.825,10.521,149.532
C07018=1130.803,308.058,-76.357,-177.828,10.520,149.533
C07019=1130.807,307.844,-76.330,-177.830,10.517,149.533
C07020=1130.810,307.631,-76.303,-177.833,10.515,149.533
C07021=1130.814,307.418,-76.275,-177.836,10.512,149.533
C07022=1130.817,307.205,-76.247,-177.838,10.510,149.533
C07023=1130.821,306.992,-76.219,-177.841,10.508,149.533
C07024=1130.825,306.744,-76.187,-177.844,10.506,149.534
C07025=1130.829,306.496,-76.156,-177.847,10.503,149.534
C07026=1130.833,306.247,-76.123,-177.850,10.501,149.534
C07027=1130.837,306.000,-76.092,-177.853,10.498,149.534
C07028=1130.841,305.752,-76.060,-177.857,10.496,149.534
C07029=1130.845,305.504,-76.027,-177.860,10.493,149.534
C07030=1130.850,305.256,-75.996,-177.863,10.490,149.535
C07031=1130.853,305.008,-75.964,-177.866,10.488,149.535
C07032=1130.858,304.760,-75.932,-177.869,10.485,149.535
C07033=1130.862,304.512,-75.900,-177.872,10.483,149.535
C07034=1130.866,304.265,-75.868,-177.875,10.480,149.535
C07035=1130.870,304.016,-75.836,-177.879,10.478,149.536
C07036=1130.874,303.768,-75.804,-177.881,10.476,149.536
C07037=1130.878,303.521,-75.772,-177.884,10.473,149.536
C07038=1130.883,303.272,-75.740,-177.887,10.470,149.536
C07039=1130.886,303.024,-75.708,-177.891,10.468,149.536
C07040=1130.891,302.777,-75.677,-177.894,10.465,149.536
C07041=1130.895,302.529,-75.645,-177.897,10.463,149.537
C07042=1130.899,302.281,-75.612,-177.900,10.460,149.537
C07043=1130.904,302.033,-75.582,-177.903,10.458,149.537
C07044=1130.907,301.785,-75.550,-177.906,10.455,149.537
C07045=1130.912,301.537,-75.518,-177.909,10.452,149.537
C07046=1130.915,301.289,-75.486,-177.913,10.450,149.538
C07047=1130.920,301.041,-75.454,-177.916,10.447,149.538
C07048=1130.924,300.794,-75.423,-177.919,10.445,149.538
C07049=1130.928,300.545,-75.391,-177.922,10.442,149.538
C07050=1130.932,300.298,-75.360,-177.925,10.440,149.538
C07051=1130.936,300.050,-75.328,-177.928,10.438,149.538
C07052=1130.940,299.802,-75.296,-177.931,10.435,149.539
C07053=1130.944,299.554,-75.266,-177.934,10.432,149.539
C07054=1130.949,299.305,-75.233,-177.937,10.430,149.539
C07055=1130.953,299.058,-75.202,-177.940,10.427,149.539
C07056=1130.957,298.809,-75.170,-177.943,10.425,149.539
C07057=1130.961,298.561,-75.139,-177.946,10.422,149.539
C07058=1130.965,298.314,-75.107,-177.950,10.419,149.540
C07059=1130.969,298.065,-75.076,-177.953,10.417,149.540
C07060=1130.973,297.818,-75.045,-177.956,10.414,149.540
C07061=1130.977,297.570,-75.013,-177.959,10.412,149.540
C07062=1130.982,297.322,-74.982,-177.962,10.409,149.540
C07063=1130.986,297.074,-74.950,-177.965,10.406,149.540
C07064=1130.990,296.826,-74.919,-177.968,10.405,149.541
C07065=1130.994,296.578,-74.887,-177.971,10.402,149.541
C07066=1130.998,296.329,-74.856,-177.974,10.400,149.541
C07067=1131.002,296.082,-74.825,-177.977,10.397,149.541
C07068=1131.006,295.833,-74.794,-177.980,10.394,149.541
C07069=1131.010,295.586,-74.762,-177.983,10.392,149.542
C07070=1131.014,295.337,-74.731,-177.987,10.389,149.542
C07071=1131.019,295.090,-74.700,-177.990,10.386,149.542
C07072=1131.022,294.876,-74.673,-177.992,10.385,149.542
C07073=1131.026,294.662,-74.646,-177.995,10.382,149.542
C07074=1131.030,294.449,-74.619,-177.998,10.380,149.542
C07075=1131.033,294.235,-74.593,-178.000,10.378,149.543
C07076=1131.036,294.022,-74.565,-178.003,10.376,149.543
C07077=1131.040,293.809,-74.538,-178.005,10.374,149.543
C07078=1131.043,293.595,-74.512,-178.008,10.371,149.543
C07079=1131.047,293.381,-74.485,-178.011,10.369,149.543
C07080=1131.051,293.133,-74.454,-178.014,10.366,149.543
C07081=1131.055,292.885,-74.422,-178.017,10.364,149.544
C07082=1131.060,292.637,-74.391,-178.020,10.361,149.544
C07083=1131.064,292.389,-74.360,-178.023,10.358,149.544
C07084=1131.068,292.141,-74.329,-178.026,10.357,149.544
C07085=1131.072,291.894,-74.299,-178.029,10.354,149.544
C07086=1131.076,291.645,-74.268,-178.032,10.352,149.545
C07087=1131.081,291.397,-74.237,-178.035,10.349,149.545
C07088=1131.084,291.149,-74.205,-178.039,10.346,149.545
C07089=1131.089,290.901,-74.174,-178.041,10.344,149.545
C07090=1131.093,290.653,-74.144,-178.045,10.341,149.545
C07091=1131.097,290.405,-74.113,-178.048,10.338,149.545
C07092=1131.101,290.157,-74.081,-178.051,10.336,149.546
C07093=1131.105,289.909,-74.050,-178.054,10.333,149.546
C07094=1131.110,289.661,-74.019,-178.057,10.331,149.546
C07095=1131.114,289.413,-73.989,-178.060,10.328,149.546
C07096=1131.118,289.165,-73.958,-178.063,10.326,149.546
C07097=1131.122,288.917,-73.927,-178.066,10.324,149.546
C07098=1131.126,288.668,-73.897,-178.069,10.321,149.547
C07099=1131.130,288.421,-73.865,-178.072,10.319,149.547
C07100=1131.134,288.173,-73.835,-178.075,10.316,149.547
C07101=1131.138,287.924,-73.803,-178.078,10.313,149.547
C07102=1131.142,287.677,-73.773,-178.081,10.311,149.547
C07103=1131.147,287.429,-73.743,-178.085,10.308,149.548
C07104=1131.151,287.180,-73.711,-178.088,10.305,149.548
C07105=1131.155,286.932,-73.681,-178.091,10.303,149.548
C07106=1131.159,286.684,-73.650,-178.094,10.300,149.548
C07107=1131.163,286.436,-73.619,-178.096,10.298,149.548
C07108=1131.167,286.188,-73.589,-178.100,10.296,149.548
C07109=1131.172,285.940,-73.558,-178.103,10.293,149.549
C07110=1131.177,285.692,-73.528,-178.106,10.291,149.549
C07111=1131.180,285.444,-73.497,-178.109,10.288,149.549
C07112=1131.185,285.195,-73.467,-178.112,10.285,149.549
C07113=1131.189,284.948,-73.437,-178.115,10.283,149.549
C07114=1131.193,284.699,-73.406,-178.118,10.280,149.550
C07115=1131.197,284.451,-73.375,-178.121,10.277,149.550
C07116=1131.201,284.203,-73.345,-178.124,10.275,149.550
C07117=1131.206,283.955,-73.314,-178.128,10.272,149.550
C07118=1131.209,283.707,-73.284,-178.130,10.270,149.550
C07119=1131.214,283.458,-73.254,-178.133,10.268,149.550
C07120=1131.218,283.211,-73.223,-178.136,10.265,149.551
C07121=1131.222,282.963,-73.193,-178.140,10.263,149.551
C07122=1131.226,282.715,-73.162,-178.143,10.260,149.551
C07123=1131.230,282.467,-73.131,-178.145,10.257,149.551
C07124=1131.234,282.218,-73.102,-178.149,10.255,149.551
C07125=1131.239,281.970,-73.071,-178.152,10.252,149.551
C07126=1131.243,281.723,-73.041,-178.155,10.250,149.552
C07127=1131.247,281.473,-73.010,-178.158,10.247,149.552
C07128=1131.251,281.260,-72.984,-178.161,10.245,149.552
C07129=1131.255,281.047,-72.959,-178.164,10.242,149.552
C07130=1131.258,280.833,-72.932,-178.167,10.240,149.552
C07131=1131.263,280.619,-72.906,-178.170,10.237,149.553
C07132=1131.265,280.406,-72.880,-178.173,10.235,149.553
C07133=1131.270,280.192,-72.854,-178.176,10.232,149.553
C07134=1131.272,279.979,-72.828,-178.180,10.230,149.553
C07135=1131.276,279.765,-72.802,-178.183,10.227,149.553
C07136=1131.280,279.517,-72.772,-178.186,10.225,149.554
C07137=1131.285,279.269,-72.742,-178.189,10.222,149.554
C07138=1131.289,279.020,-72.711,-178.193,10.219,149.554
C07139=1131.293,278.772,-72.681,-178.196,10.216,149.554
C07140=1131.297,278.524,-72.651,-178.200,10.213,149.554
C07141=1131.302,278.276,-72.622,-178.203,10.210,149.555
C07142=1131.306,278.028,-72.591,-178.206,10.208,149.555
C07143=1131.310,277.780,-72.561,-178.210,10.204,149.555
C07144=1131.314,277.532,-72.531,-178.213,10.202,149.555
C07145=1131.318,277.283,-72.501,-178.216,10.199,149.555
C07146=1131.322,277.035,-72.471,-178.219,10.196,149.555
C07147=1131.327,276.787,-72.441,-178.223,10.193,149.556
C07148=1131.331,276.538,-72.412,-178.226,10.190,149.556
C07149=1131.335,276.290,-72.381,-178.229,10.188,149.556
C07150=1131.340,276.042,-72.352,-178.232,10.185,149.556
C07151=1131.344,275.794,-72.322,-178.236,10.182,149.556
C07152=1131.348,275.546,-72.292,-178.239,10.179,149.557
C07153=1131.353,275.298,-72.262,-178.242,10.177,149.557
C07154=1131.357,275.049,-72.232,-178.245,10.174,149.557
C07155=1131.361,274.802,-72.202,-178.249,10.171,149.557
C07156=1131.365,274.554,-72.173,-178.252,10.169,149.557
C07157=1131.369,274.305,-72.143,-178.254,10.166,149.557
C07158=1131.374,274.057,-72.113,-178.257,10.163,149.557
C07159=1131.378,273.809,-72.083,-178.261,10.161,149.558
C07160=1131.382,273.561,-72.054,-178.264,10.158,149.558
C07161=1131.386,273.313,-72.024,-178.267,10.155,149.558
C07162=1131.390,273.064,-71.995,-178.270,10.152,149.558
C07163=1131.394,272.817,-71.965,-178.272,10.150,149.558
C07164=1131.398,272.568,-71.935,-178.275,10.147,149.558
C07165=1131.403,272.320,-71.905,-178.278,10.144,149.558
C07166=1131.407,272.071,-71.876,-178.282,10.142,149.559
C07167=1131.412,271.823,-71.846,-178.285,10.139,149.559
C07168=1131.416,271.575,-71.817,-178.288,10.136,149.559
C07169=1131.420,271.327,-71.787,-178.291,10.133,149.559
C07170=1131.424,271.078,-71.758,-178.293,10.131,149.559
C07171=1131.428,270.830,-71.728,-178.296,10.129,149.559
C07172=1131.432,270.583,-71.698,-178.299,10.126,149.559
C07173=1131.436,270.334,-71.669,-178.302,10.123,149.559
C07174=1131.441,270.086,-71.639,-178.304,10.121,149.559
C07175=1131.445,269.838,-71.610,-178.307,10.118,149.560
C07176=1131.449,269.589,-71.580,-178.310,10.116,149.560
C07177=1131.453,269.341,-71.551,-178.313,10.113,149.560
C07178=1131.457,269.093,-71.522,-178.315,10.111,149.560
C07179=1131.462,268.845,-71.492,-178.318,10.108,149.560
C07180=1131.466,268.596,-71.463,-178.320,10.106,149.560
C07181=1131.471,268.348,-71.434,-178.323,10.103,149.560
C07182=1131.475,268.100,-71.405,-178.326,10.100,149.560
C07183=1131.479,267.852,-71.375,-178.328,10.098,149.560
C07184=1131.483,267.638,-71.350,-178.330,10.096,149.560
C07185=1131.486,267.424,-71.324,-178.333,10.094,149.560
C07186=1131.490,267.210,-71.299,-178.335,10.092,149.560
C07187=1131.494,266.996,-71.274,-178.337,10.090,149.561
C07188=1131.498,266.783,-71.249,-178.339,10.088,149.561
C07189=1131.501,266.568,-71.223,-178.342,10.086,149.561
C07190=1131.505,266.355,-71.198,-178.343,10.084,149.561
C07191=1131.509,266.141,-71.173,-178.346,10.082,149.561
C07192=1131.513,265.893,-71.144,-178.348,10.080,149.561
C07193=1131.517,265.644,-71.114,-178.351,10.077,149.561
C07194=1131.521,265.396,-71.085,-178.353,10.075,149.561
C07195=1131.526,265.148,-71.057,-178.356,10.072,149.561
C07196=1131.530,264.900,-71.027,-178.358,10.070,149.561
C07197=1131.535,264.651,-70.998,-178.360,10.068,149.561
C07198=1131.538,264.403,-70.969,-178.363,10.065,149.561
C07199=1131.542,264.155,-70.940,-178.367,10.062,149.562
C07200=1131.547,263.906,-70.911,-178.371,10.059,149.562
C07201=1131.551,263.659,-70.882,-178.375,10.056,149.562
C07202=1131.556,263.411,-70.852,-178.379,10.053,149.563
C07203=1131.560,263.162,-70.823,-178.383,10.049,149.563
C07204=1131.564,262.914,-70.795,-178.387,10.046,149.563
C07205=1131.568,262.666,-70.765,-178.390,10.043,149.563
C07206=1131.573,262.417,-70.737,-178.394,10.040,149.564
C07207=1131.577,262.169,-70.707,-178.398,10.037,149.564
C07208=1131.581,261.920,-70.679,-178.402,10.034,149.564
C07209=1131.585,261.672,-70.650,-178.406,10.030,149.564
C07210=1131.590,261.424,-70.621,-178.409,10.028,149.564
C07211=1131.594,261.176,-70.592,-178.413,10.024,149.565
C07212=1131.599,260.927,-70.563,-178.416,10.021,149.565
C07213=1131.602,260.679,-70.534,-178.419,10.018,149.565
C07214=1131.607,260.431,-70.506,-178.423,10.015,149.565
C07215=1131.611,260.182,-70.476,-178.426,10.012,149.565
C07216=1131.615,259.934,-70.448,-178.430,10.009,149.565
C07217=1131.620,259.686,-70.419,-178.434,10.006,149.566
C07218=1131.624,259.437,-70.390,-178.437,10.003,149.566
C07219=1131.628,259.189,-70.362,-178.440,10.000,149.566
C07220=1131.633,258.941,-70.333,-178.443,9.996,149.566
C07221=1131.637,258.693,-70.305,-178.446,9.994,149.566
C07222=1131.641,258.444,-70.276,-178.450,9.990,149.566
C07223=1131.646,258.196,-70.247,-178.453,9.988,149.566
C07224=1131.650,257.948,-70.219,-178.456,9.985,149.566
C07225=1131.654,257.699,-70.190,-178.459,9.982,149.567
C07226=1131.658,257.451,-70.162,-178.463,9.979,149.567
C07227=1131.663,257.203,-70.133,-178.465,9.976,149.567
C07228=1131.667,256.954,-70.104,-178.468,9.973,149.567
C07229=1131.671,256.706,-70.076,-178.471,9.970,149.567
C07230=1131.676,256.457,-70.047,-178.474,9.967,149.567
C07231=1131.680,256.209,-70.019,-178.477,9.965,149.567
C07232=1131.684,255.961,-69.990,-178.480,9.962,149.567
C07233=1131.688,255.713,-69.962,-178.479,9.961,149.567
C07234=1131.693,255.465,-69.933,-178.478,9.960,149.566
C07235=1131.697,255.216,-69.905,-178.477,9.960,149.566
C07236=1131.701,254.967,-69.877,-178.477,9.959,149.566
C07237=1131.705,254.720,-69.848,-178.477,9.958,149.566
C07238=1131.710,254.471,-69.819,-178.477,9.957,149.565
C07239=1131.714,254.223,-69.792,-178.478,9.956,149.565
C07240=1131.718,254.009,-69.767,-178.478,9.955,149.565
C07241=1131.721,253.794,-69.742,-178.478,9.954,149.565
C07242=1131.725,253.580,-69.718,-178.480,9.953,149.565
C07243=1131.729,253.367,-69.693,-178.481,9.951,149.565
C07244=1131.733,253.153,-69.668,-178.483,9.950,149.565
C07245=1131.737,252.939,-69.644,-178.484,9.948,149.565
C07246=1131.740,252.725,-69.620,-178.486,9.946,149.565
C07247=1131.744,252.511,-69.595,-178.487,9.945,149.565
C07248=1131.749,252.263,-69.567,-178.491,9.942,149.565
C07249=1131.752,252.014,-69.539,-178.494,9.940,149.565
C07250=1131.758,251.766,-69.510,-178.497,9.937,149.566
C07251=1131.761,251.518,-69.482,-178.500,9.934,149.566
C07252=1131.765,251.269,-69.453,-178.504,9.931,149.566
C07253=1131.770,251.021,-69.425,-178.508,9.928,149.566
C07254=1131.774,250.773,-69.397,-178.512,9.925,149.567
C07255=1131.779,250.525,-69.369,-178.517,9.921,149.567
C07256=1131.782,250.276,-69.340,-178.522,9.917,149.567
C07257=1131.787,250.028,-69.313,-178.527,9.914,149.568
C07258=1131.791,249.779,-69.284,-178.532,9.910,149.568
C07259=1131.796,249.531,-69.256,-178.537,9.906,149.569
C07260=1131.799,249.283,-69.228,-178.544,9.901,149.569
C07261=1131.804,249.035,-69.200,-178.549,9.896,149.570
C07262=1131.808,248.785,-69.172,-178.556,9.892,149.570
C07263=1131.813,248.537,-69.144,-178.563,9.887,149.571
C07264=1131.817,248.289,-69.116,-178.570,9.881,149.571
C07265=1131.822,248.041,-69.088,-178.577,9.876,149.572
C07266=1131.825,247.792,-69.060,-178.584,9.870,149.573
C07267=1131.830,247.544,-69.033,-178.592,9.864,149.573
C07268=1131.834,247.296,-69.005,-178.596,9.860,149.574
C07269=1131.839,247.047,-68.976,-178.597,9.858,149.573
C07270=1131.844,246.798,-68.949,-178.599,9.856,149.573
C07271=1131.847,246.550,-68.921,-178.600,9.854,149.573
